IF (NOT(Brusa2_Tx.hton_NoPP_StopTx_Timer.Q) = TRUE) THEN
	ActAC_Rx_Timer(IN := NOT(ActAC_Rx.q_NewData), PT := T#5S);
	ActErr_Rx_Timer(IN := NOT(NLG2_ActErr_Rx.q_NewData), PT := T#5S);
	ActInt_Rx_Timer(IN := NOT(NLG2_ActInt_Rx.q_NewData), PT := T#5S);
	ActLim_Rx_Timer(IN := NOT(NLG2_ActLim_Rx.q_NewData), PT := T#5S);
	ActPlug_Rx_Timer(IN := NOT(NLG2_ActPlug_Rx.q_NewData), PT := T#5S);
	IF (ActAC_Rx_Timer.Q = TRUE AND ActErr_Rx_Timer.Q = TRUE AND ActInt_Rx_Timer.Q = TRUE AND
		ActLim_Rx_Timer.Q = TRUE AND ActPlug_Rx_Timer.Q = TRUE									) THEN
		CommsLoss	:=	TRUE;
	ELSE
		CommsLoss	:=	FALSE;
	END_IF
END_IF

Brusa2_RxConversion();

END_PROGRAM

// Application/UserCode/Brusa/Brusa2_Comms/Brusa2_RxConversion_1
PROGRAM Brusa2_RxConversion_1
VAR
ACVoltL1Act		:	UINT;
	ACVoltL2Act		:	UINT;
	ACVoltL3Act		:	UINT;
	ACCurrL1Act		:	SINT;
	ACCurrL2Act		:	SINT;
	ACCurrL3Act		:	SINT;
	ACPowTotAct		:	UINT;
	MaxTempAct		:	INT;
	TempCon			:	INT;
	DCHVAhAct			:	REAL;
	DCHVVoltAct			:	REAL;
	DCHVCurrAct			:	REAL;
	ACCurrMaxAct		:	REAL;
	ACCurrHWAvl			:	REAL;
	ACCurrMaxCP			:	REAL;
	TempCoolPlate		:	INT;		
END_VAR

ACVoltL1Act	:=	USINT_TO_UINT(Brusa2_Rx.ACVoltL1Act_Rx) * 2;
ACVoltL2Act	:=	USINT_TO_UINT(Brusa2_Rx.ACVoltL2Act_Rx) * 2;
ACVoltL3Act	:=	USINT_TO_UINT(Brusa2_Rx.ACVoltL3Act_Rx) * 2;
ACCurrL1Act	:=	USINT_TO_SINT(Brusa2_Rx.ACCurrL1Act_Rx) - 127;
ACCurrL2Act	:=	USINT_TO_SINT(Brusa2_Rx.ACCurrL2Act_Rx) - 127;
ACCurrL3Act	:=	USINT_TO_SINT(Brusa2_Rx.ACCurrL3Act_Rx) - 127;
ACPowTotAct	:=	USINT_TO_UINT(Brusa2_Rx.ACPowTotAct_Rx) * 100;
MaxTempAct	:=	USINT_TO_INT(Brusa2_Rx.MaxTempAct_Rx) - 50;
TempCon		:=	USINT_TO_INT(Brusa2_Rx.TempCon_Rx) - 50;
DCHVAhAct		:=	UINT_TO_REAL(Brusa2_Rx.DCHVAhAct_Rx) * 0.01;
DCHVVoltAct		:=	UINT_TO_REAL(Brusa2_Rx.DCHVVoltAct_Rx) * 0.1;
DCHVCurrAct		:=	UINT_TO_REAL(Brusa2_Rx.DCHVCurrAct_Rx) * 0.1 - 100;
ACCurrMaxAct	:=	UINT_TO_REAL(Brusa2_Rx.ACCurrMaxAct_Rx) * 0.1 -100;
ACCurrHWAvl		:=	USINT_TO_REAL(Brusa2_Rx.ACCurrHWAvl_Rx) * 0.5;
ACCurrMaxCP		:=	UINT_TO_REAL(Brusa2_Rx.ACCurrMaxCP_Rx) * 0.1;
TempCoolPlate	:=	USINT_TO_INT(Brusa2_Rx.TempCoolPlate_Rx) - 50;

END_PROGRAM

// Application/UserCode/Brusa/Brusa2_Comms/Brusa2_Tx_1
PROGRAM Brusa2_Tx_1

VAR
	DenLim_Tx				:	EPEC_CANVXD.Msg;
	hu8_DenLim_Tx0			:	BYTE;
	hu8_DenLim_Tx2			:	BYTE;
	hu8_DenLim_Tx4			:	BYTE;
	hu8_DenLim_Tx6			:	BYTE;
	hton_Transmit_Timer		:	TON;
	hton_NoPP_StopTx_Timer	:	TON;
	StopBroadcast			:	BOOL;
	C_VentilRq				: 	BOOL;
END_VAR


Brusa2_TxConversion();

StopBroadcast	:=	(NOT(Brusa1_Rx.S_ProximityDet)(* AND DI_q_VehicleKL15_DI = FALSE*));
hton_NoPP_StopTx_Timer(IN := StopBroadcast, PT := T#1S);

// Brusa2_Control.C_Clr_Err	:= FALSE;
hu8_DenLim_Tx0	:=	UINT_TO_USINT(SHR(Brusa2_TxConversion.DCHVVoltLimMax_Tx, 8)) + SHL(BOOL_TO_USINT(C_VentilRq), 5) +
					SHL(BOOL_TO_USINT(Brusa.S_Unlock), 6) + SHL(BOOL_TO_USINT(Brusa.S_ErrClr), 7);
hu8_DenLim_Tx2	:=	(UINT_TO_USINT(SHR(Brusa2_TxConversion.DCHVCurrLimMax_Tx, 8)) AND 2#00000111) + SHL(Brusa.S_StateDem, 5);
hu8_DenLim_Tx4	:=	(UINT_TO_USINT(SHR(Brusa2_TxConversion.ACCurrLimMax_Tx, 8)) AND 2#00000111) + SHL(Brusa.LEDDem, 4);
//hu8_DenLim_Tx6	:=	(UINT_TO_USINT(SHR(Brusa2_TxConversion.ACPhaseShift_Tx, 8)) AND 2#00001111) + SHL(BOOL_TO_USINT(Brusa2_Rx.C_EnPhaseShift), 4);

DenLim_Tx.ID		:=	16#711;
DenLim_Tx.Data[0]	:=	hu8_DenLim_Tx0;
DenLim_Tx.Data[1]	:=	UINT_TO_USINT(Brusa2_TxConversion.DCHVVoltLimMax_Tx);
DenLim_Tx.Data[2]	:=	hu8_DenLim_Tx2;
DenLim_Tx.Data[3]	:=	UINT_TO_USINT(Brusa2_TxConversion.DCHVCurrLimMax_Tx);
DenLim_Tx.Data[4]	:=	hu8_DenLim_Tx4;
DenLim_Tx.Data[5]	:=	UINT_TO_USINT(Brusa2_TxConversion.ACCurrLimMax_Tx);
DenLim_Tx.Data[6]	:=	hu8_DenLim_Tx6;
DenLim_Tx.Data[7]	:=	UINT_TO_USINT(Brusa2_TxConversion.ACPhaseShift_Tx);
DenLim_Tx.Len		:=	8;



hton_Transmit_Timer(IN := NOT(hton_Transmit_Timer.Q), PT := T#90MS);
IF (hton_Transmit_Timer.Q = TRUE AND NOT(hton_NoPP_StopTx_Timer.Q) = TRUE) THEN
	G_CAN3_Channel.SendMessage(i_pMSG:=ADR(DenLim_Tx));
END_IF

END_PROGRAM

// Application/UserCode/Brusa/Brusa2_Comms/Brusa2_TxConversion_1
PROGRAM Brusa2_TxConversion_1
VAR
		DCHVVoltLimMax_Tx	:	UINT;
		DCHVCurrLimMax_Tx	:	UINT;
		ACCurrLimMax_Tx		:	UINT;
		ACPhaseShift_Tx		:	UINT;
END_VAR

//r2
DCHVVoltLimMax_Tx	:=	REAL_TO_UINT(Brusa.S_DCHVVoltLimMax / 0.1);
DCHVCurrLimMax_Tx	:=	REAL_TO_UINT((Brusa.S_DCHVCurrLimMax - 102.4) / 0.1);
ACCurrLimMax_Tx		:=	REAL_TO_UINT((Brusa.S_ACCurrLimMax - 102.4) / 0.1);
//ACPhaseShift_Tx		:=	REAL_TO_UINT(Brusa2_Control.ACPhaseShift / 0.1);

END_PROGRAM

// Application/UserCode/CAN Function Blocks/CAN1/Callback_Receive_CAN1_1
FUNCTION_BLOCK Callback_Receive_CAN1_1 IMPLEMENTS
EPEC_CANVXD.IReceiveCallback
VAR_INPUT	
END_VAR
VAR_OUTPUT
END_VAR
VAR
END_VAR

METHOD Receive
VAR_INPUT
	(* Pointer to the CAN message *)
	i_pMsg	: POINTER TO EPEC_CANVXD.Msg;
	(* User specific argument. This is set in AddCOBID i_Argument. *)
	i_Argument	: DWORD;
END_VAR
VAR
	t_pRxMessage : POINTER TO t_CANReceive;
END_VAR


t_pRxMessage				:=	i_Argument;
t_pRxMessage^.q_NewDataRxed	:=	TRUE;
t_pRxMessage^.Data			:=	i_pMsg^.Data;
t_pRxMessage^.ID			:=	i_pMsg^.ID;
t_pRxMessage^.Len			:=	i_pMsg^.Len;
END_METHOD

END_FUNCTION_BLOCK

// Application/UserCode/CAN Function Blocks/CAN1/Receive_CAN1_EXD_1
FUNCTION_BLOCK Receive_CAN1_EXD_1
VAR_INPUT
	u32_COBID	:	DWORD;
END_VAR
VAR_OUTPUT
	q_NewData	:	BOOL;
	au8_Data	:	ARRAY [0..7] OF BYTE;
	u8_Length	:	BYTE;
END_VAR
VAR
	hq_Initialise	:	BOOL	:=	FALSE;
	ht_RxMessage	:	t_CANReceive;
	ht_MsgRx		:	Callback_Receive_CAN1;
END_VAR



IF (hq_Initialise = FALSE) THEN
	(*
	(*11 bit*)
	G_CAN1_Channel.AddCOBID(i_CobId := u32_COBID,
							i_itfCallback := ht_RxMessage,
							i_Argument := ADR(ht_RxMessage));
	*)
	(*29 bit*)
	G_CAN1_Channel.AddCOBID(i_CobId := u32_COBID OR EPEC_CANVXD.MASK_29BIT,
							i_itfCallback := ht_MsgRx,
							i_Argument := ADR(ht_RxMessage));
	G_CAN1_Channel.SetMask(i_CobID := u32_COBID OR EPEC_CANVXD.MASK_29BIT, i_Mask := (*16#0CFF0211 OR 16#0C010305 OR*) EPEC_CANVXD.MASK_29BIT);

	hq_Initialise	:=	TRUE;
END_IF


IF (ht_RxMessage.q_NewDataRxed = TRUE) THEN
	au8_Data	:=	ht_RxMessage.Data;
	u8_Length	:=	ht_RxMessage.Len;
	q_NewData	:=	TRUE;
	ht_RxMessage.q_NewDataRxed	:=	FALSE;
ELSE
	q_NewData	:=	FALSE;
END_IF

END_FUNCTION_BLOCK

// Application/UserCode/CAN Function Blocks/CAN1/Receive_CAN1_EXD_28bit_1
FUNCTION_BLOCK Receive_CAN1_EXD_28bit_1
VAR_INPUT
	u32_COBID	:	DWORD;
END_VAR
VAR_OUTPUT
	q_NewData	:	BOOL;
	au8_Data	:	ARRAY [0..7] OF BYTE;
	u8_Length	:	BYTE;
END_VAR
VAR
	hq_Initialise	:	BOOL	:=	FALSE;
	ht_RxMessage	:	t_CANReceive;
	ht_MsgRx		:	Callback_Receive_CAN1;
END_VAR



IF (hq_Initialise = FALSE) THEN
	(*
	(*11 bit*)
	G_CAN1_Channel.AddCOBID(i_CobId := u32_COBID,
							i_itfCallback := ht_RxMessage,
							i_Argument := ADR(ht_RxMessage));
	*)
	(*29 bit*)
	G_CAN1_Channel.AddCOBID(i_CobId := u32_COBID OR EPEC_CANVXD.MASK_29BIT,
							i_itfCallback := ht_MsgRx,
							i_Argument := ADR(ht_RxMessage));
	G_CAN1_Channel.SetMask(i_CobID := u32_COBID OR EPEC_CANVXD.MASK_29BIT, i_Mask := 16#0CFF0211 OR 16#0C010305 (*OR EPEC_CANVXD.MASK_29BIT*));

	hq_Initialise	:=	TRUE;
END_IF


IF (ht_RxMessage.q_NewDataRxed = TRUE) THEN
	au8_Data	:=	ht_RxMessage.Data;
	u8_Length	:=	ht_RxMessage.Len;
	q_NewData	:=	TRUE;
	ht_RxMessage.q_NewDataRxed	:=	FALSE;
ELSE
	q_NewData	:=	FALSE;
END_IF

END_FUNCTION_BLOCK

// Application/UserCode/CAN Function Blocks/CAN1/Receive_CAN1_STD_1
FUNCTION_BLOCK Receive_CAN1_STD_1
VAR_INPUT
	u32_COBID	:	DWORD;
END_VAR
VAR_OUTPUT
	q_NewData	:	BOOL;
	au8_Data	:	ARRAY [0..7] OF BYTE;
	u8_Length	:	BYTE;
END_VAR
VAR
	hq_Initialise	:	BOOL	:=	FALSE;
	ht_RxMessage	:	t_CANReceive;
	ht_MsgRx		:	Callback_Receive_CAN1;
END_VAR



IF (hq_Initialise = FALSE) THEN
	
	(*11 bit*)
	G_CAN1_Channel.AddCOBID(i_CobId := u32_COBID,
							i_itfCallback := ht_MsgRx,
							i_Argument := ADR(ht_RxMessage));
	(*
	(*29 bit*)
	G_CAN1_Channel.AddCOBID(i_CobId := u32_COBID OR EPEC_CANVXD.MASK_29BIT,
							i_itfCallback := ht_MsgRx,
							i_Argument := ADR(ht_RxMessage));
*)	(*G_CAN1_Channel.SetMask(i_CobID := u32_COBID OR EPEC_CANVXD.MASK_29BIT, i_Mask := 16#0C009000 OR EPEC_CANVXD.MASK_29BIT);
*)
	hq_Initialise	:=	TRUE;
END_IF


IF (ht_RxMessage.q_NewDataRxed = TRUE) THEN
	au8_Data	:=	ht_RxMessage.Data;
	u8_Length	:=	ht_RxMessage.Len;
	q_NewData	:=	TRUE;
	ht_RxMessage.q_NewDataRxed	:=	FALSE;
ELSE
	q_NewData	:=	FALSE;
END_IF

END_FUNCTION_BLOCK

// Application/UserCode/CAN Function Blocks/CAN2/Callback_Receive_CAN2_1
FUNCTION_BLOCK Callback_Receive_CAN2_1 IMPLEMENTS
EPEC_CANVXD.IReceiveCallback
VAR_INPUT	
END_VAR
VAR_OUTPUT
END_VAR
VAR
END_VAR

METHOD Receive
VAR_INPUT
	(* Pointer to the CAN message *)
	i_pMsg	: POINTER TO EPEC_CANVXD.Msg;
	(* User specific argument. This is set in AddCOBID i_Argument. *)
	i_Argument	: DWORD;
END_VAR
VAR
	t_pRxMessage : POINTER TO t_CANReceive;
END_VAR


t_pRxMessage				:=	i_Argument;
t_pRxMessage^.q_NewDataRxed	:=	TRUE;
t_pRxMessage^.Data			:=	i_pMsg^.Data;
t_pRxMessage^.ID			:=	i_pMsg^.ID;
t_pRxMessage^.Len			:=	i_pMsg^.Len;
END_METHOD

END_FUNCTION_BLOCK

// Application/UserCode/CAN Function Blocks/CAN2/Receive_CAN2_EXD_1
FUNCTION_BLOCK Receive_CAN2_EXD_1
VAR_INPUT
	u32_COBID	:	DWORD;
END_VAR
VAR_OUTPUT
	q_NewData	:	BOOL;
	au8_Data	:	ARRAY [0..7] OF BYTE;
	u8_Length	:	BYTE;
END_VAR
VAR
	hq_Initialise	:	BOOL	:=	FALSE;
	ht_RxMessage	:	t_CANReceive;
	ht_MsgRx		:	Callback_Receive_CAN1;
END_VAR



IF (hq_Initialise = FALSE) THEN
	(*
	IF (u32_COBID > 16#7FF) THEN
		(*29 bit*)
		;
	ELSE
		(*11 bit*)
		;
	END_IF
	*)
	(*
	(*11 bit*)
	G_CAN2_Channel.AddCOBID(i_CobId := u32_COBID,
							i_itfCallback := ht_RxMessage,
							i_Argument := ADR(ht_RxMessage));
	*)
	(*29 bit*)
	G_CAN2_Channel.AddCOBID(i_CobId := u32_COBID OR EPEC_CANVXD.MASK_29BIT,
							i_itfCallback := ht_MsgRx,
							i_Argument := ADR(ht_RxMessage));
	(*G_CAN2_Channel.SetMask(i_CobID := u32_COBID OR EPEC_CANVXD.MASK_29BIT, i_Mask := 16#0C009000 OR EPEC_CANVXD.MASK_29BIT);
*)
	hq_Initialise	:=	TRUE;
END_IF


IF (ht_RxMessage.q_NewDataRxed = TRUE) THEN
	au8_Data	:=	ht_RxMessage.Data;
	u8_Length	:=	ht_RxMessage.Len;
	q_NewData	:=	TRUE;
	ht_RxMessage.q_NewDataRxed	:=	FALSE;
ELSE
	q_NewData	:=	FALSE;
END_IF

END_FUNCTION_BLOCK

// Application/UserCode/CAN Function Blocks/CAN2/Receive_CAN2_STD_1
FUNCTION_BLOCK Receive_CAN2_STD_1
VAR_INPUT
	u32_COBID	:	DWORD;
END_VAR
VAR_OUTPUT
	q_NewData	:	BOOL;
	au8_Data	:	ARRAY [0..7] OF BYTE;
	u8_Length	:	BYTE;
END_VAR
VAR
	hq_Initialise	:	BOOL	:=	FALSE;
	ht_RxMessage	:	t_CANReceive;
	ht_MsgRx		:	Callback_Receive_CAN1;
END_VAR



IF (hq_Initialise = FALSE) THEN
	(*
	IF (u32_COBID > 16#7FF) THEN
		(*29 bit*)
		;
	ELSE
		(*11 bit*)
		;
	END_IF
	*)
	
	(*11 bit*)
	G_CAN2_Channel.AddCOBID(i_CobId := u32_COBID,
							i_itfCallback := ht_MsgRx,
							i_Argument := ADR(ht_RxMessage));
	(*
	(*29 bit*)
	G_CAN2_Channel.AddCOBID(i_CobId := u32_COBID OR EPEC_CANVXD.MASK_29BIT,
							i_itfCallback := ht_MsgRx,
							i_Argument := ADR(ht_RxMessage));
*)	(*G_CAN2_Channel.SetMask(i_CobID := u32_COBID OR EPEC_CANVXD.MASK_29BIT, i_Mask := 16#0C009000 OR EPEC_CANVXD.MASK_29BIT);
*)
	hq_Initialise	:=	TRUE;
END_IF


IF (ht_RxMessage.q_NewDataRxed = TRUE) THEN
	au8_Data	:=	ht_RxMessage.Data;
	u8_Length	:=	ht_RxMessage.Len;
	q_NewData	:=	TRUE;
	ht_RxMessage.q_NewDataRxed	:=	FALSE;
ELSE
	q_NewData	:=	FALSE;
END_IF

END_FUNCTION_BLOCK

// Application/UserCode/CAN Function Blocks/CAN3/Callback_Receive_CAN3_1
FUNCTION_BLOCK Callback_Receive_CAN3_1 IMPLEMENTS
EPEC_CANVXD.IReceiveCallback
VAR_INPUT	
END_VAR
VAR_OUTPUT
END_VAR
VAR
END_VAR

METHOD Receive
VAR_INPUT
	(* Pointer to the CAN message *)
	i_pMsg	: POINTER TO EPEC_CANVXD.Msg;
	(* User specific argument. This is set in AddCOBID i_Argument. *)
	i_Argument	: DWORD;
END_VAR
VAR
	t_pRxMessage : POINTER TO t_CANReceive;
END_VAR


t_pRxMessage				:=	i_Argument;
t_pRxMessage^.q_NewDataRxed	:=	TRUE;
t_pRxMessage^.Data			:=	i_pMsg^.Data;
t_pRxMessage^.ID			:=	i_pMsg^.ID;
t_pRxMessage^.Len			:=	i_pMsg^.Len;
END_METHOD

END_FUNCTION_BLOCK

// Application/UserCode/CAN Function Blocks/CAN3/Receive_CAN3_EXD_1
FUNCTION_BLOCK Receive_CAN3_EXD_1
VAR_INPUT
	u32_COBID	:	DWORD;
END_VAR
VAR_OUTPUT
	q_NewData	:	BOOL;
	au8_Data	:	ARRAY [0..7] OF BYTE;
	u8_Length	:	BYTE;
END_VAR
VAR
	hq_Initialise	:	BOOL	:=	FALSE;
	ht_RxMessage	:	t_CANReceive;
	ht_MsgRx		:	Callback_Receive_CAN1;
END_VAR



IF (hq_Initialise = FALSE) THEN
	(*
	IF (u32_COBID > 16#7FF) THEN
		(*29 bit*)
		;
	ELSE
		(*11 bit*)
		;
	END_IF
	*)
	(*
	(*11 bit*)
	G_CAN3_Channel.AddCOBID(i_CobId := u32_COBID,
							i_itfCallback := ht_RxMessage,
							i_Argument := ADR(ht_RxMessage));
	*)
	(*29 bit*)
	G_CAN3_Channel.AddCOBID(i_CobId := u32_COBID OR EPEC_CANVXD.MASK_29BIT,
							i_itfCallback := ht_MsgRx,
							i_Argument := ADR(ht_RxMessage));
	G_CAN3_Channel.SetMask(i_CobID := u32_COBID OR EPEC_CANVXD.MASK_29BIT, (*i_Mask := 16#0C009000 OR*) EPEC_CANVXD.MASK_29BIT);

	hq_Initialise	:=	TRUE;
END_IF


IF (ht_RxMessage.q_NewDataRxed = TRUE) THEN
	au8_Data	:=	ht_RxMessage.Data;
	u8_Length	:=	ht_RxMessage.Len;
	q_NewData	:=	TRUE;
	ht_RxMessage.q_NewDataRxed	:=	FALSE;
ELSE
	q_NewData	:=	FALSE;
END_IF

END_FUNCTION_BLOCK

// Application/UserCode/CAN Function Blocks/CAN3/Receive_CAN3_EXD_28bit_1
FUNCTION_BLOCK Receive_CAN3_EXD_28bit_1
VAR_INPUT
	u32_COBID	:	DWORD;
END_VAR
VAR_OUTPUT
	q_NewData	:	BOOL;
	au8_Data	:	ARRAY [0..7] OF BYTE;
	u8_Length	:	BYTE;
END_VAR
VAR
	hq_Initialise	:	BOOL	:=	FALSE;
	ht_RxMessage	:	t_CANReceive;
	ht_MsgRx		:	Callback_Receive_CAN1;
END_VAR



IF (hq_Initialise = FALSE) THEN
	(*
	IF (u32_COBID > 16#7FF) THEN
		(*29 bit*)
		;
	ELSE
		(*11 bit*)
		;
	END_IF
	*)
	(*
	(*11 bit*)
	G_CAN3_Channel.AddCOBID(i_CobId := u32_COBID,
							i_itfCallback := ht_RxMessage,
							i_Argument := ADR(ht_RxMessage));
	*)
	(*29 bit*)
	G_CAN3_Channel.AddCOBID(i_CobId := u32_COBID OR EPEC_CANVXD.MASK_29BIT,
							i_itfCallback := ht_MsgRx,
							i_Argument := ADR(ht_RxMessage));
	G_CAN3_Channel.SetMask(i_CobID := u32_COBID OR EPEC_CANVXD.MASK_29BIT, i_Mask := 16#0C010305);

	hq_Initialise	:=	TRUE;
END_IF


IF (ht_RxMessage.q_NewDataRxed = TRUE) THEN
	au8_Data	:=	ht_RxMessage.Data;
	u8_Length	:=	ht_RxMessage.Len;
	q_NewData	:=	TRUE;
	ht_RxMessage.q_NewDataRxed	:=	FALSE;
ELSE
	q_NewData	:=	FALSE;
END_IF

END_FUNCTION_BLOCK

// Application/UserCode/CAN Function Blocks/CAN3/Receive_CAN3_STD_1
FUNCTION_BLOCK Receive_CAN3_STD_1
VAR_INPUT
	u32_COBID	:	DWORD;
END_VAR
VAR_OUTPUT
	q_NewData	:	BOOL;
	au8_Data	:	ARRAY [0..7] OF BYTE;
	u8_Length	:	BYTE;
END_VAR
VAR
	hq_Initialise	:	BOOL	:=	FALSE;
	ht_RxMessage	:	t_CANReceive;
	ht_MsgRx		:	Callback_Receive_CAN1;
END_VAR



IF (hq_Initialise = FALSE) THEN
	(*
	IF (u32_COBID > 16#7FF) THEN
		(*29 bit*)
		;
	ELSE
		(*11 bit*)
		;
	END_IF
	*)
	
	(*11 bit*)
	G_CAN3_Channel.AddCOBID(i_CobId := u32_COBID,
							i_itfCallback := ht_MsgRx,
							i_Argument := ADR(ht_RxMessage));
	(*
	(*29 bit*)
	G_CAN3_Channel.AddCOBID(i_CobId := u32_COBID OR EPEC_CANVXD.MASK_29BIT,
							i_itfCallback := ht_MsgRx,
							i_Argument := ADR(ht_RxMessage));
*)	(*G_CAN3_Channel.SetMask(i_CobID := u32_COBID OR EPEC_CANVXD.MASK_29BIT, i_Mask := 16#0C009000 OR EPEC_CANVXD.MASK_29BIT);
*)
	hq_Initialise	:=	TRUE;
END_IF


IF (ht_RxMessage.q_NewDataRxed = TRUE) THEN
	au8_Data	:=	ht_RxMessage.Data;
	u8_Length	:=	ht_RxMessage.Len;
	q_NewData	:=	TRUE;
	ht_RxMessage.q_NewDataRxed	:=	FALSE;
ELSE
	q_NewData	:=	FALSE;
END_IF

END_FUNCTION_BLOCK

// Application/UserCode/CAN Function Blocks/CAN4/Callback_Receive_CAN4_1
FUNCTION_BLOCK Callback_Receive_CAN4_1 IMPLEMENTS
EPEC_CANVXD.IReceiveCallback
VAR_INPUT	
END_VAR
VAR_OUTPUT
END_VAR
VAR
END_VAR

METHOD Receive
VAR_INPUT
	(* Pointer to the CAN message *)
	i_pMsg	: POINTER TO EPEC_CANVXD.Msg;
	(* User specific argument. This is set in AddCOBID i_Argument. *)
	i_Argument	: DWORD;
END_VAR
VAR
	t_pRxMessage : POINTER TO t_CANReceive;
END_VAR


t_pRxMessage				:=	i_Argument;
t_pRxMessage^.q_NewDataRxed	:=	TRUE;
t_pRxMessage^.Data			:=	i_pMsg^.Data;
t_pRxMessage^.ID			:=	i_pMsg^.ID;
t_pRxMessage^.Len			:=	i_pMsg^.Len;
END_METHOD

END_FUNCTION_BLOCK

// Application/UserCode/CAN Function Blocks/CAN4/Receive_CAN4_EXD_1
FUNCTION_BLOCK Receive_CAN4_EXD_1
VAR_INPUT
	u32_COBID	:	DWORD;
END_VAR
VAR_OUTPUT
	q_NewData	:	BOOL;
	au8_Data	:	ARRAY [0..7] OF BYTE;
	u8_Length	:	BYTE;
END_VAR
VAR
	hq_Initialise	:	BOOL	:=	FALSE;
	ht_RxMessage	:	t_CANReceive;
	ht_MsgRx		:	Callback_Receive_CAN1;
END_VAR



IF (hq_Initialise = FALSE) THEN
	(*
	IF (u32_COBID > 16#7FF) THEN
		(*29 bit*)
		;
	ELSE
		(*11 bit*)
		;
	END_IF
	*)
	(*
	(*11 bit*)
	G_CAN4_Channel.AddCOBID(i_CobId := u32_COBID,
							i_itfCallback := ht_RxMessage,
							i_Argument := ADR(ht_RxMessage));
	*)
	(*29 bit*)
	G_CAN4_Channel.AddCOBID(i_CobId := u32_COBID OR EPEC_CANVXD.MASK_29BIT,
							i_itfCallback := ht_MsgRx,
							i_Argument := ADR(ht_RxMessage));
	G_CAN4_Channel.SetMask(i_CobID := u32_COBID OR EPEC_CANVXD.MASK_29BIT, i_Mask := 16#18FEF1F2 OR EPEC_CANVXD.MASK_29BIT);

	hq_Initialise	:=	TRUE;
END_IF


IF (ht_RxMessage.q_NewDataRxed = TRUE) THEN
	au8_Data	:=	ht_RxMessage.Data;
	u8_Length	:=	ht_RxMessage.Len;
	q_NewData	:=	TRUE;
	ht_RxMessage.q_NewDataRxed	:=	FALSE;
ELSE
	q_NewData	:=	FALSE;
END_IF

END_FUNCTION_BLOCK

// Application/UserCode/CAN Function Blocks/CAN4/Receive_CAN4_STD_1
FUNCTION_BLOCK Receive_CAN4_STD_1
VAR_INPUT
	u32_COBID	:	DWORD;
END_VAR
VAR_OUTPUT
	q_NewData	:	BOOL;
	au8_Data	:	ARRAY [0..7] OF BYTE;
	u8_Length	:	BYTE;
END_VAR
VAR
	hq_Initialise	:	BOOL	:=	FALSE;
	ht_RxMessage	:	t_CANReceive;
	ht_MsgRx		:	Callback_Receive_CAN1;
END_VAR



IF (hq_Initialise = FALSE) THEN
	(*
	IF (u32_COBID > 16#7FF) THEN
		(*29 bit*)
		;
	ELSE
		(*11 bit*)
		;
	END_IF
	*)
	
	(*11 bit*)
	G_CAN4_Channel.AddCOBID(i_CobId := u32_COBID,
							i_itfCallback := ht_MsgRx,
							i_Argument := ADR(ht_RxMessage));
	(*
	(*29 bit*)
	G_CAN4_Channel.AddCOBID(i_CobId := u32_COBID OR EPEC_CANVXD.MASK_29BIT,
							i_itfCallback := ht_MsgRx,
							i_Argument := ADR(ht_RxMessage));
*)	(*G_CAN4_Channel.SetMask(i_CobID := u32_COBID OR EPEC_CANVXD.MASK_29BIT, i_Mask := 16#0C009000 OR EPEC_CANVXD.MASK_29BIT);
*)
	hq_Initialise	:=	TRUE;
END_IF


IF (ht_RxMessage.q_NewDataRxed = TRUE) THEN
	au8_Data	:=	ht_RxMessage.Data;
	u8_Length	:=	ht_RxMessage.Len;
	q_NewData	:=	TRUE;
	ht_RxMessage.q_NewDataRxed	:=	FALSE;
ELSE
	q_NewData	:=	FALSE;
END_IF

END_FUNCTION_BLOCK

// Application/UserCode/Main Program/RealTimeClock
PROGRAM RealTimeClock

VAR
	RTC_0: rtc;
	Timesky: DATE_AND_TIME := DT#2021-10-29-17:31:0;
	today: DATE_AND_TIME;
	a1870: DATE_AND_TIME := DT#1970-1-1-0:0:0;
END_VAR

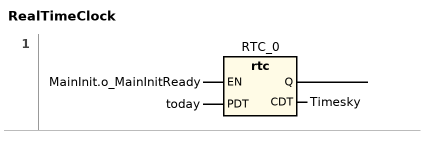
// NETWORK 1
RTC_0(EN := MainInit.o_MainInitReady, PDT := today, CDT => Timesky); // rtc

END_PROGRAM

// Application/UserCode/HMI/Data to or For HMI/BMS_to_HMI_1
PROGRAM BMS_to_HMI_1
VAR
	ht_CAN4_DD0_Tx	:	EPEC_CANVXD.Msg;
	ht_CAN4_DD1_Tx	:	EPEC_CANVXD.Msg;
	ht_CAN4_DD2_Tx	:	EPEC_CANVXD.Msg;
	ht_CAN4_DD3_Tx	:	EPEC_CANVXD.Msg;
	ht_CAN4_DD4_Tx	:	EPEC_CANVXD.Msg;
	ht_CAN4_DD5_Tx	:	EPEC_CANVXD.Msg;
	ht_CAN4_DD6_Tx	:	EPEC_CANVXD.Msg;
	ht_CAN4_DD7_Tx	:	EPEC_CANVXD.Msg;
	ht_CAN4_DD8_Tx	:	EPEC_CANVXD.Msg;
	ht_CAN4_DD9_Tx	:	EPEC_CANVXD.Msg;
	ht_CAN4_DDA_Tx	:	EPEC_CANVXD.Msg;
	ht_CAN4_DDB_Tx	:	EPEC_CANVXD.Msg;
	ht_CAN4_DDC_Tx	:	EPEC_CANVXD.Msg;
	ht_CAN4_DDD_Tx	:	EPEC_CANVXD.Msg;
	ht_CAN4_ADD0_Tx	:	EPEC_CANVXD.Msg;
	ht_CAN4_ADD1_Tx	:	EPEC_CANVXD.Msg;
	ht_CAN4_ADD2_Tx	:	EPEC_CANVXD.Msg;
	ht_CAN4_ADD3_Tx	:	EPEC_CANVXD.Msg;
	ht_CAN4_ADD4_Tx	:	EPEC_CANVXD.Msg;
	ht_CAN4_ADD5_Tx	:	EPEC_CANVXD.Msg;
	ht_CAN4_ADD6_Tx	:	EPEC_CANVXD.Msg;
	ht_CAN4_ADD7_Tx	:	EPEC_CANVXD.Msg;
	ht_CAN4_ADD8_Tx	:	EPEC_CANVXD.Msg;
	ht_CAN4_ADD9_Tx	:	EPEC_CANVXD.Msg;
	ht_CAN4_ADDA_Tx	:	EPEC_CANVXD.Msg;
	ht_CAN4_ADDB_Tx	:	EPEC_CANVXD.Msg;
	ht_CAN4_ADDC_Tx	:	EPEC_CANVXD.Msg;
	ht_CAN4_ADDD_Tx	:	EPEC_CANVXD.Msg;
	hton_MessageSend_Timer	:	TON;
	
	Tx_Timer	:	TON;
	
END_VAR

//Send raw BMS Data to HMI CAN#4
(*BMS1*)
ht_CAN4_DD0_Tx.ID		:=	16#181000DD OR EPEC_CANVXD.MASK_29BIT;
ht_CAN4_DD0_Tx.Data[0]	:=	OrionBMS1_Rx.OrionBMS1_6B0_Rx.au8_Data[0];
ht_CAN4_DD0_Tx.Data[1]	:=	OrionBMS1_Rx.OrionBMS1_6B0_Rx.au8_Data[1];
ht_CAN4_DD0_Tx.Data[2]	:=	OrionBMS1_Rx.OrionBMS1_6B0_Rx.au8_Data[2];
ht_CAN4_DD0_Tx.Data[3]	:=	OrionBMS1_Rx.OrionBMS1_6B0_Rx.au8_Data[3];
ht_CAN4_DD0_Tx.Data[4]	:=	OrionBMS1_Rx.OrionBMS1_6B0_Rx.au8_Data[4];
ht_CAN4_DD0_Tx.Data[5]	:=	OrionBMS1_Rx.OrionBMS1_6B0_Rx.au8_Data[5];		
ht_CAN4_DD0_Tx.Data[6]	:=	OrionBMS1_Rx.OrionBMS1_6B0_Rx.au8_Data[6];	
ht_CAN4_DD0_Tx.Data[7]	:=	OrionBMS1_Rx.OrionBMS1_6B0_Rx.au8_Data[7];		
ht_CAN4_DD0_Tx.Len		:=	8;

ht_CAN4_DD1_Tx.ID		:=	16#181001DD OR EPEC_CANVXD.MASK_29BIT;
ht_CAN4_DD1_Tx.Data[0]	:=	OrionBMS1_Rx.OrionBMS1_6B1_Rx.au8_Data[0];
ht_CAN4_DD1_Tx.Data[1]	:=	OrionBMS1_Rx.OrionBMS1_6B1_Rx.au8_Data[1];
ht_CAN4_DD1_Tx.Data[2]	:=	OrionBMS1_Rx.OrionBMS1_6B1_Rx.au8_Data[2];
ht_CAN4_DD1_Tx.Data[3]	:=	OrionBMS1_Rx.OrionBMS1_6B1_Rx.au8_Data[3];
ht_CAN4_DD1_Tx.Data[4]	:=	OrionBMS1_Rx.OrionBMS1_6B1_Rx.au8_Data[4];
ht_CAN4_DD1_Tx.Data[5]	:=	OrionBMS1_Rx.OrionBMS1_6B1_Rx.au8_Data[5];		
ht_CAN4_DD1_Tx.Data[6]	:=	OrionBMS1_Rx.OrionBMS1_6B1_Rx.au8_Data[6];	
ht_CAN4_DD1_Tx.Data[7]	:=	OrionBMS1_Rx.OrionBMS1_6B1_Rx.au8_Data[7];		
ht_CAN4_DD1_Tx.Len		:=	8;

ht_CAN4_DD2_Tx.ID		:=	16#181002DD OR EPEC_CANVXD.MASK_29BIT;
ht_CAN4_DD2_Tx.Data[0]	:=	OrionBMS1_Rx.OrionBMS1_6B2_Rx.au8_Data[0];
ht_CAN4_DD2_Tx.Data[1]	:=	OrionBMS1_Rx.OrionBMS1_6B2_Rx.au8_Data[1];
ht_CAN4_DD2_Tx.Data[2]	:=	OrionBMS1_Rx.OrionBMS1_6B2_Rx.au8_Data[2];
ht_CAN4_DD2_Tx.Data[3]	:=	OrionBMS1_Rx.OrionBMS1_6B2_Rx.au8_Data[3];
ht_CAN4_DD2_Tx.Data[4]	:=	OrionBMS1_Rx.OrionBMS1_6B2_Rx.au8_Data[4];
ht_CAN4_DD2_Tx.Data[5]	:=	OrionBMS1_Rx.OrionBMS1_6B2_Rx.au8_Data[5];		
ht_CAN4_DD2_Tx.Data[6]	:=	OrionBMS1_Rx.OrionBMS1_6B2_Rx.au8_Data[6];	
ht_CAN4_DD2_Tx.Data[7]	:=	OrionBMS1_Rx.OrionBMS1_6B2_Rx.au8_Data[7];		
ht_CAN4_DD2_Tx.Len		:=	8;

ht_CAN4_DD3_Tx.ID		:=	16#181003DD OR EPEC_CANVXD.MASK_29BIT;
ht_CAN4_DD3_Tx.Data[0]	:=	OrionBMS1_Rx.OrionBMS1_6B3_Rx.au8_Data[0];
ht_CAN4_DD3_Tx.Data[1]	:=	OrionBMS1_Rx.OrionBMS1_6B3_Rx.au8_Data[1];
ht_CAN4_DD3_Tx.Data[2]	:=	OrionBMS1_Rx.OrionBMS1_6B3_Rx.au8_Data[2];
ht_CAN4_DD3_Tx.Data[3]	:=	OrionBMS1_Rx.OrionBMS1_6B3_Rx.au8_Data[3];
ht_CAN4_DD3_Tx.Data[4]	:=	OrionBMS1_Rx.OrionBMS1_6B3_Rx.au8_Data[4];
ht_CAN4_DD3_Tx.Data[5]	:=	OrionBMS1_Rx.OrionBMS1_6B3_Rx.au8_Data[5];		
ht_CAN4_DD3_Tx.Data[6]	:=	OrionBMS1_Rx.OrionBMS1_6B3_Rx.au8_Data[6];	
ht_CAN4_DD3_Tx.Data[7]	:=	OrionBMS1_Rx.OrionBMS1_6B3_Rx.au8_Data[7];		
ht_CAN4_DD3_Tx.Len		:=	8;

ht_CAN4_DD4_Tx.ID		:=	16#181004DD OR EPEC_CANVXD.MASK_29BIT;
ht_CAN4_DD4_Tx.Data[0]	:=	OrionBMS1_Rx.OrionBMS1_6B4_Rx.au8_Data[0];
ht_CAN4_DD4_Tx.Data[1]	:=	OrionBMS1_Rx.OrionBMS1_6B4_Rx.au8_Data[1];
ht_CAN4_DD4_Tx.Data[2]	:=	OrionBMS1_Rx.OrionBMS1_6B4_Rx.au8_Data[2];
ht_CAN4_DD4_Tx.Data[3]	:=	OrionBMS1_Rx.OrionBMS1_6B4_Rx.au8_Data[3];
ht_CAN4_DD4_Tx.Data[4]	:=	OrionBMS1_Rx.OrionBMS1_6B4_Rx.au8_Data[4];
ht_CAN4_DD4_Tx.Data[5]	:=	OrionBMS1_Rx.OrionBMS1_6B4_Rx.au8_Data[5];		
ht_CAN4_DD4_Tx.Data[6]	:=	OrionBMS1_Rx.OrionBMS1_6B4_Rx.au8_Data[6];	
ht_CAN4_DD4_Tx.Data[7]	:=	OrionBMS1_Rx.OrionBMS1_6B4_Rx.au8_Data[7];		
ht_CAN4_DD4_Tx.Len		:=	8;

ht_CAN4_DD5_Tx.ID		:=	16#181005DD OR EPEC_CANVXD.MASK_29BIT;
ht_CAN4_DD5_Tx.Data[0]	:=	OrionBMS1_Rx.OrionBMS1_6B5_Rx.au8_Data[0];
ht_CAN4_DD5_Tx.Data[1]	:=	OrionBMS1_Rx.OrionBMS1_6B5_Rx.au8_Data[1];
ht_CAN4_DD5_Tx.Data[2]	:=	OrionBMS1_Rx.OrionBMS1_6B5_Rx.au8_Data[2];
ht_CAN4_DD5_Tx.Data[3]	:=	OrionBMS1_Rx.OrionBMS1_6B5_Rx.au8_Data[3];
ht_CAN4_DD5_Tx.Data[4]	:=	OrionBMS1_Rx.OrionBMS1_6B5_Rx.au8_Data[4];
ht_CAN4_DD5_Tx.Data[5]	:=	OrionBMS1_Rx.OrionBMS1_6B5_Rx.au8_Data[5];		
ht_CAN4_DD5_Tx.Data[6]	:=	OrionBMS1_Rx.OrionBMS1_6B5_Rx.au8_Data[6];	
ht_CAN4_DD5_Tx.Data[7]	:=	OrionBMS1_Rx.OrionBMS1_6B5_Rx.au8_Data[7];		
ht_CAN4_DD5_Tx.Len		:=	8;

ht_CAN4_DD6_Tx.ID		:=	16#181006DD OR EPEC_CANVXD.MASK_29BIT;
ht_CAN4_DD6_Tx.Data[0]	:=	OrionBMS1_Rx.OrionBMS1_6B6_Rx.au8_Data[0];
ht_CAN4_DD6_Tx.Data[1]	:=	OrionBMS1_Rx.OrionBMS1_6B6_Rx.au8_Data[1];
ht_CAN4_DD6_Tx.Data[2]	:=	OrionBMS1_Rx.OrionBMS1_6B6_Rx.au8_Data[2];
ht_CAN4_DD6_Tx.Data[3]	:=	OrionBMS1_Rx.OrionBMS1_6B6_Rx.au8_Data[3];
ht_CAN4_DD6_Tx.Data[4]	:=	OrionBMS1_Rx.OrionBMS1_6B6_Rx.au8_Data[4];
ht_CAN4_DD6_Tx.Data[5]	:=	OrionBMS1_Rx.OrionBMS1_6B6_Rx.au8_Data[5];		
ht_CAN4_DD6_Tx.Data[6]	:=	OrionBMS1_Rx.OrionBMS1_6B6_Rx.au8_Data[6];	
ht_CAN4_DD6_Tx.Data[7]	:=	OrionBMS1_Rx.OrionBMS1_6B6_Rx.au8_Data[7];		
ht_CAN4_DD6_Tx.Len		:=	8;

ht_CAN4_DD7_Tx.ID		:=	16#181007DD OR EPEC_CANVXD.MASK_29BIT;
ht_CAN4_DD7_Tx.Data[0]	:=	OrionBMS1_Rx.OrionBMS1_6B7_Rx.au8_Data[0];
ht_CAN4_DD7_Tx.Data[1]	:=	OrionBMS1_Rx.OrionBMS1_6B7_Rx.au8_Data[1];
ht_CAN4_DD7_Tx.Data[2]	:=	OrionBMS1_Rx.OrionBMS1_6B7_Rx.au8_Data[2];
ht_CAN4_DD7_Tx.Data[3]	:=	OrionBMS1_Rx.OrionBMS1_6B7_Rx.au8_Data[3];
ht_CAN4_DD7_Tx.Data[4]	:=	OrionBMS1_Rx.OrionBMS1_6B7_Rx.au8_Data[4];
ht_CAN4_DD7_Tx.Data[5]	:=	OrionBMS1_Rx.OrionBMS1_6B7_Rx.au8_Data[5];		
ht_CAN4_DD7_Tx.Data[6]	:=	OrionBMS1_Rx.OrionBMS1_6B7_Rx.au8_Data[6];	
ht_CAN4_DD7_Tx.Data[7]	:=	OrionBMS1_Rx.OrionBMS1_6B7_Rx.au8_Data[7];		
ht_CAN4_DD7_Tx.Len		:=	8;

ht_CAN4_DD8_Tx.ID		:=	16#181008DD OR EPEC_CANVXD.MASK_29BIT;
ht_CAN4_DD8_Tx.Data[0]	:=	OrionBMS1_Rx.OrionBMS1_6B8_Rx.au8_Data[0];
ht_CAN4_DD8_Tx.Data[1]	:=	OrionBMS1_Rx.OrionBMS1_6B8_Rx.au8_Data[1];
ht_CAN4_DD8_Tx.Data[2]	:=	OrionBMS1_Rx.OrionBMS1_6B8_Rx.au8_Data[2];
ht_CAN4_DD8_Tx.Data[3]	:=	OrionBMS1_Rx.OrionBMS1_6B8_Rx.au8_Data[3];
ht_CAN4_DD8_Tx.Data[4]	:=	OrionBMS1_Rx.OrionBMS1_6B8_Rx.au8_Data[4];
ht_CAN4_DD8_Tx.Data[5]	:=	OrionBMS1_Rx.OrionBMS1_6B8_Rx.au8_Data[5];		
ht_CAN4_DD8_Tx.Data[6]	:=	OrionBMS1_Rx.OrionBMS1_6B8_Rx.au8_Data[6];	
ht_CAN4_DD8_Tx.Data[7]	:=	OrionBMS1_Rx.OrionBMS1_6B8_Rx.au8_Data[7];		
ht_CAN4_DD8_Tx.Len		:=	8;

ht_CAN4_DD9_Tx.ID		:=	16#181009DD OR EPEC_CANVXD.MASK_29BIT;
ht_CAN4_DD9_Tx.Data[0]	:=	OrionBMS1_Rx.OrionBMS1_6B9_Rx.au8_Data[0];
ht_CAN4_DD9_Tx.Data[1]	:=	OrionBMS1_Rx.OrionBMS1_6B9_Rx.au8_Data[1];
ht_CAN4_DD9_Tx.Data[2]	:=	OrionBMS1_Rx.OrionBMS1_6B9_Rx.au8_Data[2];
ht_CAN4_DD9_Tx.Data[3]	:=	OrionBMS1_Rx.OrionBMS1_6B9_Rx.au8_Data[3];
ht_CAN4_DD9_Tx.Data[4]	:=	OrionBMS1_Rx.OrionBMS1_6B9_Rx.au8_Data[4];
ht_CAN4_DD9_Tx.Data[5]	:=	OrionBMS1_Rx.OrionBMS1_6B9_Rx.au8_Data[5];		
ht_CAN4_DD9_Tx.Data[6]	:=	OrionBMS1_Rx.OrionBMS1_6B9_Rx.au8_Data[6];	
ht_CAN4_DD9_Tx.Data[7]	:=	OrionBMS1_Rx.OrionBMS1_6B9_Rx.au8_Data[7];		
ht_CAN4_DD9_Tx.Len		:=	8;

ht_CAN4_DDA_Tx.ID		:=	16#18100ADD OR EPEC_CANVXD.MASK_29BIT;
ht_CAN4_DDA_Tx.Data[0]	:=	OrionBMS1_Rx.OrionBMS1_6BA_Rx.au8_Data[0];
ht_CAN4_DDA_Tx.Data[1]	:=	OrionBMS1_Rx.OrionBMS1_6BA_Rx.au8_Data[1];
ht_CAN4_DDA_Tx.Data[2]	:=	OrionBMS1_Rx.OrionBMS1_6BA_Rx.au8_Data[2];
ht_CAN4_DDA_Tx.Data[3]	:=	OrionBMS1_Rx.OrionBMS1_6BA_Rx.au8_Data[3];
ht_CAN4_DDA_Tx.Data[4]	:=	OrionBMS1_Rx.OrionBMS1_6BA_Rx.au8_Data[4];
ht_CAN4_DDA_Tx.Data[5]	:=	OrionBMS1_Rx.OrionBMS1_6BA_Rx.au8_Data[5];		
ht_CAN4_DDA_Tx.Data[6]	:=	OrionBMS1_Rx.OrionBMS1_6BA_Rx.au8_Data[6];	
ht_CAN4_DDA_Tx.Data[7]	:=	OrionBMS1_Rx.OrionBMS1_6BA_Rx.au8_Data[7];		
ht_CAN4_DDA_Tx.Len		:=	8;

ht_CAN4_DDB_Tx.ID		:=	16#18100BDD OR EPEC_CANVXD.MASK_29BIT;
ht_CAN4_DDB_Tx.Data[0]	:=	OrionBMS1_Rx.OrionBMS1_6BB_Rx.au8_Data[0];
ht_CAN4_DDB_Tx.Data[1]	:=	OrionBMS1_Rx.OrionBMS1_6BB_Rx.au8_Data[1];
ht_CAN4_DDB_Tx.Data[2]	:=	OrionBMS1_Rx.OrionBMS1_6BB_Rx.au8_Data[2];
ht_CAN4_DDB_Tx.Data[3]	:=	OrionBMS1_Rx.OrionBMS1_6BB_Rx.au8_Data[3];
ht_CAN4_DDB_Tx.Data[4]	:=	OrionBMS1_Rx.OrionBMS1_6BB_Rx.au8_Data[4];
ht_CAN4_DDB_Tx.Data[5]	:=	OrionBMS1_Rx.OrionBMS1_6BB_Rx.au8_Data[5];		
ht_CAN4_DDB_Tx.Data[6]	:=	OrionBMS1_Rx.OrionBMS1_6BB_Rx.au8_Data[6];	
ht_CAN4_DDB_Tx.Data[7]	:=	OrionBMS1_Rx.OrionBMS1_6BB_Rx.au8_Data[7];		
ht_CAN4_DDB_Tx.Len		:=	8;

ht_CAN4_DDC_Tx.ID		:=	16#18100CDD OR EPEC_CANVXD.MASK_29BIT;
ht_CAN4_DDC_Tx.Data[0]	:=	OrionBMS1_Rx.OrionBMS1_6BC_Rx.au8_Data[0];
ht_CAN4_DDC_Tx.Data[1]	:=	OrionBMS1_Rx.OrionBMS1_6BC_Rx.au8_Data[1];
ht_CAN4_DDC_Tx.Data[2]	:=	OrionBMS1_Rx.OrionBMS1_6BC_Rx.au8_Data[2];
ht_CAN4_DDC_Tx.Data[3]	:=	OrionBMS1_Rx.OrionBMS1_6BC_Rx.au8_Data[3];
ht_CAN4_DDC_Tx.Data[4]	:=	OrionBMS1_Rx.OrionBMS1_6BC_Rx.au8_Data[4];
ht_CAN4_DDC_Tx.Data[5]	:=	OrionBMS1_Rx.OrionBMS1_6BC_Rx.au8_Data[5];		
ht_CAN4_DDC_Tx.Data[6]	:=	OrionBMS1_Rx.OrionBMS1_6BC_Rx.au8_Data[6];	
ht_CAN4_DDC_Tx.Data[7]	:=	OrionBMS1_Rx.OrionBMS1_6BC_Rx.au8_Data[7];		
ht_CAN4_DDC_Tx.Len		:=	8;

ht_CAN4_DDD_Tx.ID		:=	16#18100DDD OR EPEC_CANVXD.MASK_29BIT;
ht_CAN4_DDD_Tx.Data[0]	:=	OrionBMS1_Rx.OrionBMS1_6BD_Rx.au8_Data[0];
ht_CAN4_DDD_Tx.Data[1]	:=	OrionBMS1_Rx.OrionBMS1_6BD_Rx.au8_Data[1];
ht_CAN4_DDD_Tx.Data[2]	:=	OrionBMS1_Rx.OrionBMS1_6BD_Rx.au8_Data[2];
ht_CAN4_DDD_Tx.Data[3]	:=	OrionBMS1_Rx.OrionBMS1_6BD_Rx.au8_Data[3];
ht_CAN4_DDD_Tx.Data[4]	:=	OrionBMS1_Rx.OrionBMS1_6BD_Rx.au8_Data[4];
ht_CAN4_DDD_Tx.Data[5]	:=	OrionBMS1_Rx.OrionBMS1_6BD_Rx.au8_Data[5];		
ht_CAN4_DDD_Tx.Data[6]	:=	OrionBMS1_Rx.OrionBMS1_6BD_Rx.au8_Data[6];	
ht_CAN4_DDD_Tx.Data[7]	:=	OrionBMS1_Rx.OrionBMS1_6BD_Rx.au8_Data[7];		
ht_CAN4_DDD_Tx.Len		:=	8;

//*BMS Slave
ht_CAN4_ADD0_Tx.ID		:=	16#182000DD OR EPEC_CANVXD.MASK_29BIT;
ht_CAN4_ADD0_Tx.Data[0]	:=	OrionBMS2_Rx.OrionBMS2_6B0_Rx.au8_Data[0];
ht_CAN4_ADD0_Tx.Data[1]	:=	OrionBMS2_Rx.OrionBMS2_6B0_Rx.au8_Data[1];
ht_CAN4_ADD0_Tx.Data[2]	:=	OrionBMS2_Rx.OrionBMS2_6B0_Rx.au8_Data[2];
ht_CAN4_ADD0_Tx.Data[3]	:=	OrionBMS2_Rx.OrionBMS2_6B0_Rx.au8_Data[3];
ht_CAN4_ADD0_Tx.Data[4]	:=	OrionBMS2_Rx.OrionBMS2_6B0_Rx.au8_Data[4];
ht_CAN4_ADD0_Tx.Data[5]	:=	OrionBMS2_Rx.OrionBMS2_6B0_Rx.au8_Data[5];		
ht_CAN4_ADD0_Tx.Data[6]	:=	OrionBMS2_Rx.OrionBMS2_6B0_Rx.au8_Data[6];	
ht_CAN4_ADD0_Tx.Data[7]	:=	OrionBMS2_Rx.OrionBMS2_6B0_Rx.au8_Data[7];		
ht_CAN4_ADD0_Tx.Len		:=	8;

ht_CAN4_ADD1_Tx.ID		:=	16#182001DD OR EPEC_CANVXD.MASK_29BIT;
ht_CAN4_ADD1_Tx.Data[0]	:=	OrionBMS2_Rx.OrionBMS2_6B1_Rx.au8_Data[0];
ht_CAN4_ADD1_Tx.Data[1]	:=	OrionBMS2_Rx.OrionBMS2_6B1_Rx.au8_Data[1];
ht_CAN4_ADD1_Tx.Data[2]	:=	OrionBMS2_Rx.OrionBMS2_6B1_Rx.au8_Data[2];
ht_CAN4_ADD1_Tx.Data[3]	:=	OrionBMS2_Rx.OrionBMS2_6B1_Rx.au8_Data[3];
ht_CAN4_ADD1_Tx.Data[4]	:=	OrionBMS2_Rx.OrionBMS2_6B1_Rx.au8_Data[4];
ht_CAN4_ADD1_Tx.Data[5]	:=	OrionBMS2_Rx.OrionBMS2_6B1_Rx.au8_Data[5];		
ht_CAN4_ADD1_Tx.Data[6]	:=	OrionBMS2_Rx.OrionBMS2_6B1_Rx.au8_Data[6];	
ht_CAN4_ADD1_Tx.Data[7]	:=	OrionBMS2_Rx.OrionBMS2_6B1_Rx.au8_Data[7];		
ht_CAN4_ADD1_Tx.Len		:=	8;

ht_CAN4_ADD2_Tx.ID		:=	16#182002DD OR EPEC_CANVXD.MASK_29BIT;
ht_CAN4_ADD2_Tx.Data[0]	:=	OrionBMS2_Rx.OrionBMS2_6B2_Rx.au8_Data[0];
ht_CAN4_ADD2_Tx.Data[1]	:=	OrionBMS2_Rx.OrionBMS2_6B2_Rx.au8_Data[1];
ht_CAN4_ADD2_Tx.Data[2]	:=	OrionBMS2_Rx.OrionBMS2_6B2_Rx.au8_Data[2];
ht_CAN4_ADD2_Tx.Data[3]	:=	OrionBMS2_Rx.OrionBMS2_6B2_Rx.au8_Data[3];
ht_CAN4_ADD2_Tx.Data[4]	:=	OrionBMS2_Rx.OrionBMS2_6B2_Rx.au8_Data[4];
ht_CAN4_ADD2_Tx.Data[5]	:=	OrionBMS2_Rx.OrionBMS2_6B2_Rx.au8_Data[5];		
ht_CAN4_ADD2_Tx.Data[6]	:=	OrionBMS2_Rx.OrionBMS2_6B2_Rx.au8_Data[6];	
ht_CAN4_ADD2_Tx.Data[7]	:=	OrionBMS2_Rx.OrionBMS2_6B2_Rx.au8_Data[7];		
ht_CAN4_ADD2_Tx.Len		:=	8;

ht_CAN4_ADD3_Tx.ID		:=	16#182003DD OR EPEC_CANVXD.MASK_29BIT;
ht_CAN4_ADD3_Tx.Data[0]	:=	OrionBMS2_Rx.OrionBMS2_6B3_Rx.au8_Data[0];
ht_CAN4_ADD3_Tx.Data[1]	:=	OrionBMS2_Rx.OrionBMS2_6B3_Rx.au8_Data[1];
ht_CAN4_ADD3_Tx.Data[2]	:=	OrionBMS2_Rx.OrionBMS2_6B3_Rx.au8_Data[2];
ht_CAN4_ADD3_Tx.Data[3]	:=	OrionBMS2_Rx.OrionBMS2_6B3_Rx.au8_Data[3];
ht_CAN4_ADD3_Tx.Data[4]	:=	OrionBMS2_Rx.OrionBMS2_6B3_Rx.au8_Data[4];
ht_CAN4_ADD3_Tx.Data[5]	:=	OrionBMS2_Rx.OrionBMS2_6B3_Rx.au8_Data[5];		
ht_CAN4_ADD3_Tx.Data[6]	:=	OrionBMS2_Rx.OrionBMS2_6B3_Rx.au8_Data[6];	
ht_CAN4_ADD3_Tx.Data[7]	:=	OrionBMS2_Rx.OrionBMS2_6B3_Rx.au8_Data[7];		
ht_CAN4_ADD3_Tx.Len		:=	8;

ht_CAN4_ADD4_Tx.ID		:=	16#182004DD OR EPEC_CANVXD.MASK_29BIT;
ht_CAN4_ADD4_Tx.Data[0]	:=	OrionBMS2_Rx.OrionBMS2_6B4_Rx.au8_Data[0];
ht_CAN4_ADD4_Tx.Data[1]	:=	OrionBMS2_Rx.OrionBMS2_6B4_Rx.au8_Data[1];
ht_CAN4_ADD4_Tx.Data[2]	:=	OrionBMS2_Rx.OrionBMS2_6B4_Rx.au8_Data[2];
ht_CAN4_ADD4_Tx.Data[3]	:=	OrionBMS2_Rx.OrionBMS2_6B4_Rx.au8_Data[3];
ht_CAN4_ADD4_Tx.Data[4]	:=	OrionBMS2_Rx.OrionBMS2_6B4_Rx.au8_Data[4];
ht_CAN4_ADD4_Tx.Data[5]	:=	OrionBMS2_Rx.OrionBMS2_6B4_Rx.au8_Data[5];		
ht_CAN4_ADD4_Tx.Data[6]	:=	OrionBMS2_Rx.OrionBMS2_6B4_Rx.au8_Data[6];	
ht_CAN4_ADD4_Tx.Data[7]	:=	OrionBMS2_Rx.OrionBMS2_6B4_Rx.au8_Data[7];		
ht_CAN4_ADD4_Tx.Len		:=	8;

ht_CAN4_ADD5_Tx.ID		:=	16#182005DD OR EPEC_CANVXD.MASK_29BIT;
ht_CAN4_ADD5_Tx.Data[0]	:=	OrionBMS2_Rx.OrionBMS2_6B5_Rx.au8_Data[0];
ht_CAN4_ADD5_Tx.Data[1]	:=	OrionBMS2_Rx.OrionBMS2_6B5_Rx.au8_Data[1];
ht_CAN4_ADD5_Tx.Data[2]	:=	OrionBMS2_Rx.OrionBMS2_6B5_Rx.au8_Data[2];
ht_CAN4_ADD5_Tx.Data[3]	:=	OrionBMS2_Rx.OrionBMS2_6B5_Rx.au8_Data[3];
ht_CAN4_ADD5_Tx.Data[4]	:=	OrionBMS2_Rx.OrionBMS2_6B5_Rx.au8_Data[4];
ht_CAN4_ADD5_Tx.Data[5]	:=	OrionBMS2_Rx.OrionBMS2_6B5_Rx.au8_Data[5];		
ht_CAN4_ADD5_Tx.Data[6]	:=	OrionBMS2_Rx.OrionBMS2_6B5_Rx.au8_Data[6];	
ht_CAN4_ADD5_Tx.Data[7]	:=	OrionBMS2_Rx.OrionBMS2_6B5_Rx.au8_Data[7];		
ht_CAN4_ADD5_Tx.Len		:=	8;

ht_CAN4_ADD6_Tx.ID		:=	16#182006DD OR EPEC_CANVXD.MASK_29BIT;
ht_CAN4_ADD6_Tx.Data[0]	:=	OrionBMS2_Rx.OrionBMS2_6B6_Rx.au8_Data[0];
ht_CAN4_ADD6_Tx.Data[1]	:=	OrionBMS2_Rx.OrionBMS2_6B6_Rx.au8_Data[1];
ht_CAN4_ADD6_Tx.Data[2]	:=	OrionBMS2_Rx.OrionBMS2_6B6_Rx.au8_Data[2];
ht_CAN4_ADD6_Tx.Data[3]	:=	OrionBMS2_Rx.OrionBMS2_6B6_Rx.au8_Data[3];
ht_CAN4_ADD6_Tx.Data[4]	:=	OrionBMS2_Rx.OrionBMS2_6B6_Rx.au8_Data[4];
ht_CAN4_ADD6_Tx.Data[5]	:=	OrionBMS2_Rx.OrionBMS2_6B6_Rx.au8_Data[5];		
ht_CAN4_ADD6_Tx.Data[6]	:=	OrionBMS2_Rx.OrionBMS2_6B6_Rx.au8_Data[6];	
ht_CAN4_ADD6_Tx.Data[7]	:=	OrionBMS2_Rx.OrionBMS2_6B6_Rx.au8_Data[7];		
ht_CAN4_ADD6_Tx.Len		:=	8;

ht_CAN4_ADD7_Tx.ID		:=	16#182007DD OR EPEC_CANVXD.MASK_29BIT;
ht_CAN4_ADD7_Tx.Data[0]	:=	OrionBMS2_Rx.OrionBMS2_6B7_Rx.au8_Data[0];
ht_CAN4_ADD7_Tx.Data[1]	:=	OrionBMS2_Rx.OrionBMS2_6B7_Rx.au8_Data[1];
ht_CAN4_ADD7_Tx.Data[2]	:=	OrionBMS2_Rx.OrionBMS2_6B7_Rx.au8_Data[2];
ht_CAN4_ADD7_Tx.Data[3]	:=	OrionBMS2_Rx.OrionBMS2_6B7_Rx.au8_Data[3];
ht_CAN4_ADD7_Tx.Data[4]	:=	OrionBMS2_Rx.OrionBMS2_6B7_Rx.au8_Data[4];
ht_CAN4_ADD7_Tx.Data[5]	:=	OrionBMS2_Rx.OrionBMS2_6B7_Rx.au8_Data[5];		
ht_CAN4_ADD7_Tx.Data[6]	:=	OrionBMS2_Rx.OrionBMS2_6B7_Rx.au8_Data[6];	
ht_CAN4_ADD7_Tx.Data[7]	:=	OrionBMS2_Rx.OrionBMS2_6B7_Rx.au8_Data[7];		
ht_CAN4_ADD7_Tx.Len		:=	8;

ht_CAN4_ADD8_Tx.ID		:=	16#182008DD OR EPEC_CANVXD.MASK_29BIT;
ht_CAN4_ADD8_Tx.Data[0]	:=	OrionBMS2_Rx.OrionBMS2_6B8_Rx.au8_Data[0];
ht_CAN4_ADD8_Tx.Data[1]	:=	OrionBMS2_Rx.OrionBMS2_6B8_Rx.au8_Data[1];
ht_CAN4_ADD8_Tx.Data[2]	:=	OrionBMS2_Rx.OrionBMS2_6B8_Rx.au8_Data[2];
ht_CAN4_ADD8_Tx.Data[3]	:=	OrionBMS2_Rx.OrionBMS2_6B8_Rx.au8_Data[3];
ht_CAN4_ADD8_Tx.Data[4]	:=	OrionBMS2_Rx.OrionBMS2_6B8_Rx.au8_Data[4];
ht_CAN4_ADD8_Tx.Data[5]	:=	OrionBMS2_Rx.OrionBMS2_6B8_Rx.au8_Data[5];		
ht_CAN4_ADD8_Tx.Data[6]	:=	OrionBMS2_Rx.OrionBMS2_6B8_Rx.au8_Data[6];	
ht_CAN4_ADD8_Tx.Data[7]	:=	OrionBMS2_Rx.OrionBMS2_6B8_Rx.au8_Data[7];		
ht_CAN4_ADD8_Tx.Len		:=	8;

ht_CAN4_ADD9_Tx.ID		:=	16#182009DD OR EPEC_CANVXD.MASK_29BIT;
ht_CAN4_ADD9_Tx.Data[0]	:=	OrionBMS2_Rx.OrionBMS2_6B9_Rx.au8_Data[0];
ht_CAN4_ADD9_Tx.Data[1]	:=	OrionBMS2_Rx.OrionBMS2_6B9_Rx.au8_Data[1];
ht_CAN4_ADD9_Tx.Data[2]	:=	OrionBMS2_Rx.OrionBMS2_6B9_Rx.au8_Data[2];
ht_CAN4_ADD9_Tx.Data[3]	:=	OrionBMS2_Rx.OrionBMS2_6B9_Rx.au8_Data[3];
ht_CAN4_ADD9_Tx.Data[4]	:=	OrionBMS2_Rx.OrionBMS2_6B9_Rx.au8_Data[4];
ht_CAN4_ADD9_Tx.Data[5]	:=	OrionBMS2_Rx.OrionBMS2_6B9_Rx.au8_Data[5];		
ht_CAN4_ADD9_Tx.Data[6]	:=	OrionBMS2_Rx.OrionBMS2_6B9_Rx.au8_Data[6];	
ht_CAN4_ADD9_Tx.Data[7]	:=	OrionBMS2_Rx.OrionBMS2_6B9_Rx.au8_Data[7];		
ht_CAN4_ADD9_Tx.Len		:=	8;

ht_CAN4_ADDA_Tx.ID		:=	16#18200ADD OR EPEC_CANVXD.MASK_29BIT;
ht_CAN4_ADDA_Tx.Data[0]	:=	OrionBMS2_Rx.OrionBMS2_6BA_Rx.au8_Data[0];
ht_CAN4_ADDA_Tx.Data[1]	:=	OrionBMS2_Rx.OrionBMS2_6BA_Rx.au8_Data[1];
ht_CAN4_ADDA_Tx.Data[2]	:=	OrionBMS2_Rx.OrionBMS2_6BA_Rx.au8_Data[2];
ht_CAN4_ADDA_Tx.Data[3]	:=	OrionBMS2_Rx.OrionBMS2_6BA_Rx.au8_Data[3];
ht_CAN4_ADDA_Tx.Data[4]	:=	OrionBMS2_Rx.OrionBMS2_6BA_Rx.au8_Data[4];
ht_CAN4_ADDA_Tx.Data[5]	:=	OrionBMS2_Rx.OrionBMS2_6BA_Rx.au8_Data[5];		
ht_CAN4_ADDA_Tx.Data[6]	:=	OrionBMS2_Rx.OrionBMS2_6BA_Rx.au8_Data[6];	
ht_CAN4_ADDA_Tx.Data[7]	:=	OrionBMS2_Rx.OrionBMS2_6BA_Rx.au8_Data[7];		
ht_CAN4_ADDA_Tx.Len		:=	8;

ht_CAN4_ADDB_Tx.ID		:=	16#18200BDD OR EPEC_CANVXD.MASK_29BIT;
ht_CAN4_ADDB_Tx.Data[0]	:=	OrionBMS2_Rx.OrionBMS2_6BB_Rx.au8_Data[0];
ht_CAN4_ADDB_Tx.Data[1]	:=	OrionBMS2_Rx.OrionBMS2_6BB_Rx.au8_Data[1];
ht_CAN4_ADDB_Tx.Data[2]	:=	OrionBMS2_Rx.OrionBMS2_6BB_Rx.au8_Data[2];
ht_CAN4_ADDB_Tx.Data[3]	:=	OrionBMS2_Rx.OrionBMS2_6BB_Rx.au8_Data[3];
ht_CAN4_ADDB_Tx.Data[4]	:=	OrionBMS2_Rx.OrionBMS2_6BB_Rx.au8_Data[4];
ht_CAN4_ADDB_Tx.Data[5]	:=	OrionBMS2_Rx.OrionBMS2_6BB_Rx.au8_Data[5];		
ht_CAN4_ADDB_Tx.Data[6]	:=	OrionBMS2_Rx.OrionBMS2_6BB_Rx.au8_Data[6];	
ht_CAN4_ADDB_Tx.Data[7]	:=	OrionBMS2_Rx.OrionBMS2_6BB_Rx.au8_Data[7];		
ht_CAN4_ADDB_Tx.Len		:=	8;

ht_CAN4_ADDC_Tx.ID		:=	16#18200CDD OR EPEC_CANVXD.MASK_29BIT;
ht_CAN4_ADDC_Tx.Data[0]	:=	OrionBMS2_Rx.OrionBMS2_6BC_Rx.au8_Data[0];
ht_CAN4_ADDC_Tx.Data[1]	:=	OrionBMS2_Rx.OrionBMS2_6BC_Rx.au8_Data[1];
ht_CAN4_ADDC_Tx.Data[2]	:=	OrionBMS2_Rx.OrionBMS2_6BC_Rx.au8_Data[2];
ht_CAN4_ADDC_Tx.Data[3]	:=	OrionBMS2_Rx.OrionBMS2_6BC_Rx.au8_Data[3];
ht_CAN4_ADDC_Tx.Data[4]	:=	OrionBMS2_Rx.OrionBMS2_6BC_Rx.au8_Data[4];
ht_CAN4_ADDC_Tx.Data[5]	:=	OrionBMS2_Rx.OrionBMS2_6BC_Rx.au8_Data[5];		
ht_CAN4_ADDC_Tx.Data[6]	:=	OrionBMS2_Rx.OrionBMS2_6BC_Rx.au8_Data[6];	
ht_CAN4_ADDC_Tx.Data[7]	:=	OrionBMS2_Rx.OrionBMS2_6BC_Rx.au8_Data[7];		
ht_CAN4_ADDC_Tx.Len		:=	8;

ht_CAN4_ADDD_Tx.ID		:=	16#18200DDD OR EPEC_CANVXD.MASK_29BIT;
ht_CAN4_ADDD_Tx.Data[0]	:=	OrionBMS2_Rx.OrionBMS2_6BD_Rx.au8_Data[0];
ht_CAN4_ADDD_Tx.Data[1]	:=	OrionBMS2_Rx.OrionBMS2_6BD_Rx.au8_Data[1];
ht_CAN4_ADDD_Tx.Data[2]	:=	OrionBMS2_Rx.OrionBMS2_6BD_Rx.au8_Data[2];
ht_CAN4_ADDD_Tx.Data[3]	:=	OrionBMS2_Rx.OrionBMS2_6BD_Rx.au8_Data[3];
ht_CAN4_ADDD_Tx.Data[4]	:=	OrionBMS2_Rx.OrionBMS2_6BD_Rx.au8_Data[4];
ht_CAN4_ADDD_Tx.Data[5]	:=	OrionBMS2_Rx.OrionBMS2_6BD_Rx.au8_Data[5];		
ht_CAN4_ADDD_Tx.Data[6]	:=	OrionBMS2_Rx.OrionBMS2_6BD_Rx.au8_Data[6];	
ht_CAN4_ADDD_Tx.Data[7]	:=	OrionBMS2_Rx.OrionBMS2_6BD_Rx.au8_Data[7];		
ht_CAN4_ADDD_Tx.Len		:=	8;



Tx_Timer(IN := NOT(Tx_Timer.Q), PT := T#1000MS);
IF (Tx_Timer.Q = TRUE) THEN
	G_CAN4_Channel.SendMessage(i_pMSG:=ADR(ht_CAN4_DD0_Tx));
	G_CAN4_Channel.SendMessage(i_pMSG:=ADR(ht_CAN4_DD1_Tx));
	G_CAN4_Channel.SendMessage(i_pMSG:=ADR(ht_CAN4_DD2_Tx));
	G_CAN4_Channel.SendMessage(i_pMSG:=ADR(ht_CAN4_DD3_Tx));
	G_CAN4_Channel.SendMessage(i_pMSG:=ADR(ht_CAN4_DD4_Tx));
	G_CAN4_Channel.SendMessage(i_pMSG:=ADR(ht_CAN4_DD5_Tx));
	G_CAN4_Channel.SendMessage(i_pMSG:=ADR(ht_CAN4_DD6_Tx));
	G_CAN4_Channel.SendMessage(i_pMSG:=ADR(ht_CAN4_DD7_Tx));
	G_CAN4_Channel.SendMessage(i_pMSG:=ADR(ht_CAN4_DD8_Tx));
	G_CAN4_Channel.SendMessage(i_pMSG:=ADR(ht_CAN4_DD9_Tx));
	G_CAN4_Channel.SendMessage(i_pMSG:=ADR(ht_CAN4_DDA_Tx));
	G_CAN4_Channel.SendMessage(i_pMSG:=ADR(ht_CAN4_DDB_Tx));
	G_CAN4_Channel.SendMessage(i_pMSG:=ADR(ht_CAN4_DDC_Tx));
	G_CAN4_Channel.SendMessage(i_pMSG:=ADR(ht_CAN4_DDD_Tx));
	G_CAN4_Channel.SendMessage(i_pMSG:=ADR(ht_CAN4_ADD0_Tx));
	G_CAN4_Channel.SendMessage(i_pMSG:=ADR(ht_CAN4_ADD1_Tx));
	G_CAN4_Channel.SendMessage(i_pMSG:=ADR(ht_CAN4_ADD2_Tx));
	G_CAN4_Channel.SendMessage(i_pMSG:=ADR(ht_CAN4_ADD3_Tx));
	G_CAN4_Channel.SendMessage(i_pMSG:=ADR(ht_CAN4_ADD4_Tx));
	G_CAN4_Channel.SendMessage(i_pMSG:=ADR(ht_CAN4_ADD5_Tx));
	G_CAN4_Channel.SendMessage(i_pMSG:=ADR(ht_CAN4_ADD6_Tx));
	G_CAN4_Channel.SendMessage(i_pMSG:=ADR(ht_CAN4_ADD7_Tx));
	G_CAN4_Channel.SendMessage(i_pMSG:=ADR(ht_CAN4_ADD8_Tx));
	G_CAN4_Channel.SendMessage(i_pMSG:=ADR(ht_CAN4_ADD9_Tx));
	G_CAN4_Channel.SendMessage(i_pMSG:=ADR(ht_CAN4_ADDA_Tx));
	G_CAN4_Channel.SendMessage(i_pMSG:=ADR(ht_CAN4_ADDB_Tx));
	G_CAN4_Channel.SendMessage(i_pMSG:=ADR(ht_CAN4_ADDC_Tx));
	G_CAN4_Channel.SendMessage(i_pMSG:=ADR(ht_CAN4_ADDD_Tx));
	
END_IF

END_PROGRAM

// Application/UserCode/HMI/Data to or For HMI/BRUSA_to_HMI_1
PROGRAM BRUSA_to_HMI_1
VAR
	ht_CAN4_7DD0_Tx	:	EPEC_CANVXD.Msg;
	ht_CAN4_7DD1_Tx	:	EPEC_CANVXD.Msg;
	ht_CAN4_7DD2_Tx: EPEC_CANVXD.msg;
	ht_CAN4_7DD3_Tx: EPEC_CANVXD.msg;
	ht_CAN4_7DD4_Tx: EPEC_CANVXD.msg;
	ht_CAN4_7DD5_Tx: EPEC_CANVXD.msg;
	ht_CAN4_7DD6_Tx: EPEC_CANVXD.msg;
	ht_CAN4_7DD7_Tx: EPEC_CANVXD.msg;
	ht_CAN4_7DD8_Tx: EPEC_CANVXD.msg;
	ht_CAN4_7DD9_Tx: EPEC_CANVXD.msg;
	ht_CAN4_7DDA_Tx: EPEC_CANVXD.msg;
	ht_CAN4_7DDB_Tx: EPEC_CANVXD.msg;
	hton_MessageSend_Timer	:	TON;
	Tx_Timer	:	TON;
	END_VAR

//called from can4_TX

//Master Brusa
ht_CAN4_7DD0_Tx.ID		:=	16#187000DD OR EPEC_CANVXD.MASK_29BIT;
ht_CAN4_7DD0_Tx.Data[0]	:=	Brusa1_Rx.ActAC_Rx.au8_Data[0];
ht_CAN4_7DD0_Tx.Data[1]	:=	Brusa1_Rx.ActAC_Rx.au8_Data[1];
ht_CAN4_7DD0_Tx.Data[2]	:=	Brusa1_Rx.ActAC_Rx.au8_Data[2];
ht_CAN4_7DD0_Tx.Data[3]	:=	Brusa1_Rx.ActAC_Rx.au8_Data[3];
ht_CAN4_7DD0_Tx.Data[4]	:=	Brusa1_Rx.ActAC_Rx.au8_Data[4];
ht_CAN4_7DD0_Tx.Data[5]	:=	Brusa1_Rx.ActAC_Rx.au8_Data[5];
ht_CAN4_7DD0_Tx.Data[6]	:=	Brusa1_Rx.ActAC_Rx.au8_Data[6];
ht_CAN4_7DD0_Tx.Data[7]	:=	Brusa1_Rx.ActAC_Rx.au8_Data[7];
ht_CAN4_7DD0_Tx.Len		:=	8;

//* Errors
ht_CAN4_7DD2_Tx.ID		:=	16#187002DD OR EPEC_CANVXD.MASK_29BIT;
ht_CAN4_7DD2_Tx.Data[0]	:=	Brusa1_Rx.ActErr_Rx.au8_Data[0];
ht_CAN4_7DD2_Tx.Data[1]	:=	Brusa1_Rx.ActErr_Rx.au8_Data[1];
ht_CAN4_7DD2_Tx.Data[2]	:=	Brusa1_Rx.ActErr_Rx.au8_Data[2];
ht_CAN4_7DD2_Tx.Data[3]	:=	Brusa1_Rx.ActErr_Rx.au8_Data[3];
ht_CAN4_7DD2_Tx.Data[4]	:=	Brusa1_Rx.ActErr_Rx.au8_Data[4];
ht_CAN4_7DD2_Tx.Data[5]	:=	Brusa1_Rx.ActErr_Rx.au8_Data[5];
ht_CAN4_7DD2_Tx.Data[6]	:=	Brusa1_Rx.ActErr_Rx.au8_Data[6];
ht_CAN4_7DD2_Tx.Data[7]	:=	Brusa1_Rx.ActErr_Rx.au8_Data[7];
ht_CAN4_7DD2_Tx.Len		:=	8;

ht_CAN4_7DD4_Tx.ID		:=	16#187004DD OR EPEC_CANVXD.MASK_29BIT;
ht_CAN4_7DD4_Tx.Data[0]	:=	Brusa1_Rx.ActInt_Rx.au8_Data[0];
ht_CAN4_7DD4_Tx.Data[1]	:=	Brusa1_Rx.ActInt_Rx.au8_Data[1];
ht_CAN4_7DD4_Tx.Data[2]	:=	Brusa1_Rx.ActInt_Rx.au8_Data[2];
ht_CAN4_7DD4_Tx.Data[3]	:=	Brusa1_Rx.ActInt_Rx.au8_Data[3];
ht_CAN4_7DD4_Tx.Data[4]	:=	Brusa1_Rx.ActInt_Rx.au8_Data[4];
ht_CAN4_7DD4_Tx.Data[5]	:=	Brusa1_Rx.ActInt_Rx.au8_Data[5];
ht_CAN4_7DD4_Tx.Data[6]	:=	Brusa1_Rx.ActInt_Rx.au8_Data[6];
ht_CAN4_7DD4_Tx.Data[7]	:=	Brusa1_Rx.ActInt_Rx.au8_Data[7];
ht_CAN4_7DD4_Tx.Len		:=	8;

ht_CAN4_7DD6_Tx.ID		:=	16#187006DD OR EPEC_CANVXD.MASK_29BIT;
ht_CAN4_7DD6_Tx.Data[0]	:=	Brusa1_Rx.ActLim_Rx.au8_Data[0];
ht_CAN4_7DD6_Tx.Data[1]	:=	Brusa1_Rx.ActLim_Rx.au8_Data[1];
ht_CAN4_7DD6_Tx.Data[2]	:=	Brusa1_Rx.ActLim_Rx.au8_Data[2];
ht_CAN4_7DD6_Tx.Data[3]	:=	Brusa1_Rx.ActLim_Rx.au8_Data[3];
ht_CAN4_7DD6_Tx.Data[4]	:=	Brusa1_Rx.ActLim_Rx.au8_Data[4];
ht_CAN4_7DD6_Tx.Data[5]	:=	Brusa1_Rx.ActLim_Rx.au8_Data[5];
ht_CAN4_7DD6_Tx.Data[6]	:=	Brusa1_Rx.ActLim_Rx.au8_Data[6];
ht_CAN4_7DD6_Tx.Data[7]	:=	Brusa1_Rx.ActLim_Rx.au8_Data[7];
ht_CAN4_7DD6_Tx.Len		:=	8;

ht_CAN4_7DD8_Tx.ID		:=	16#187008DD OR EPEC_CANVXD.MASK_29BIT;
ht_CAN4_7DD8_Tx.Data[0]	:=	Brusa1_Rx.ActPlug_Rx.au8_Data[0];
ht_CAN4_7DD8_Tx.Data[1]	:=	Brusa1_Rx.ActPlug_Rx.au8_Data[1];
ht_CAN4_7DD8_Tx.Data[2]	:=	Brusa1_Rx.ActPlug_Rx.au8_Data[2];
ht_CAN4_7DD8_Tx.Data[3]	:=	Brusa1_Rx.ActPlug_Rx.au8_Data[3];
ht_CAN4_7DD8_Tx.Data[4]	:=	Brusa1_Rx.ActPlug_Rx.au8_Data[4];
ht_CAN4_7DD8_Tx.Data[5]	:=	Brusa1_Rx.ActPlug_Rx.au8_Data[5];
ht_CAN4_7DD8_Tx.Data[6]	:=	Brusa1_Rx.ActPlug_Rx.au8_Data[6];
ht_CAN4_7DD8_Tx.Data[7]	:=	Brusa1_Rx.ActPlug_Rx.au8_Data[7];
ht_CAN4_7DD8_Tx.Len		:=	8;

ht_CAN4_7DDA_Tx.ID		:=	16#18700ADD OR EPEC_CANVXD.MASK_29BIT;
ht_CAN4_7DDA_Tx.Data[0]	:=	Brusa1_Tx.DenLim_Tx.Data[0];
ht_CAN4_7DDA_Tx.Data[1]	:=	Brusa1_Tx.DenLim_Tx.Data[1];
ht_CAN4_7DDA_Tx.Data[2]	:=	Brusa1_Tx.DenLim_Tx.Data[2];
ht_CAN4_7DDA_Tx.Data[3]	:=	Brusa1_Tx.DenLim_Tx.Data[3];
ht_CAN4_7DDA_Tx.Data[4]	:=	Brusa1_Tx.DenLim_Tx.Data[4];
ht_CAN4_7DDA_Tx.Data[5]	:=	Brusa1_Tx.DenLim_Tx.Data[5];
ht_CAN4_7DDA_Tx.Data[6]	:=	Brusa1_Tx.DenLim_Tx.Data[6];
ht_CAN4_7DDA_Tx.Data[7]	:=	Brusa1_Tx.DenLim_Tx.Data[7];
ht_CAN4_7DDA_Tx.Len		:=	8;



//Slave Brusa
ht_CAN4_7DD1_Tx.ID		:=	16#187001DD OR EPEC_CANVXD.MASK_29BIT;
ht_CAN4_7DD1_Tx.Data[0]	:=	Brusa2_Rx.ActAC_Rx.au8_Data[0];
ht_CAN4_7DD1_Tx.Data[1]	:=	Brusa2_Rx.ActAC_Rx.au8_Data[1];
ht_CAN4_7DD1_Tx.Data[2]	:=	Brusa2_Rx.ActAC_Rx.au8_Data[2];
ht_CAN4_7DD1_Tx.Data[3]	:=	Brusa2_Rx.ActAC_Rx.au8_Data[3];
ht_CAN4_7DD1_Tx.Data[4]	:=	Brusa2_Rx.ActAC_Rx.au8_Data[4];
ht_CAN4_7DD1_Tx.Data[5]	:=	Brusa2_Rx.ActAC_Rx.au8_Data[5];
ht_CAN4_7DD1_Tx.Data[6]	:=	Brusa2_Rx.ActAC_Rx.au8_Data[6];
ht_CAN4_7DD1_Tx.Data[7]	:=	Brusa2_Rx.ActAC_Rx.au8_Data[7];
ht_CAN4_7DD1_Tx.Len		:=	8;

ht_CAN4_7DD3_Tx.ID		:=	16#187003DD OR EPEC_CANVXD.MASK_29BIT;
ht_CAN4_7DD3_Tx.Data[0]	:=	Brusa2_Rx.NLG2_ActErr_Rx.au8_Data[0];
ht_CAN4_7DD3_Tx.Data[1]	:=	Brusa2_Rx.NLG2_ActErr_Rx.au8_Data[1];
ht_CAN4_7DD3_Tx.Data[2]	:=	Brusa2_Rx.NLG2_ActErr_Rx.au8_Data[2];
ht_CAN4_7DD3_Tx.Data[3]	:=	Brusa2_Rx.NLG2_ActErr_Rx.au8_Data[3];
ht_CAN4_7DD3_Tx.Data[4]	:=	Brusa2_Rx.NLG2_ActErr_Rx.au8_Data[4];
ht_CAN4_7DD3_Tx.Data[5]	:=	Brusa2_Rx.NLG2_ActErr_Rx.au8_Data[5];
ht_CAN4_7DD3_Tx.Data[6]	:=	Brusa2_Rx.NLG2_ActErr_Rx.au8_Data[6];
ht_CAN4_7DD3_Tx.Data[7]	:=	Brusa2_Rx.NLG2_ActErr_Rx.au8_Data[7];
ht_CAN4_7DD3_Tx.Len		:=	8;

ht_CAN4_7DD5_Tx.ID		:=	16#187005DD OR EPEC_CANVXD.MASK_29BIT;
ht_CAN4_7DD5_Tx.Data[0]	:=	Brusa2_Rx.NLG2_ActInt_Rx.au8_Data[0];
ht_CAN4_7DD5_Tx.Data[1]	:=	Brusa2_Rx.NLG2_ActInt_Rx.au8_Data[1];
ht_CAN4_7DD5_Tx.Data[2]	:=	Brusa2_Rx.NLG2_ActInt_Rx.au8_Data[2];
ht_CAN4_7DD5_Tx.Data[3]	:=	Brusa2_Rx.NLG2_ActInt_Rx.au8_Data[3];
ht_CAN4_7DD5_Tx.Data[4]	:=	Brusa2_Rx.NLG2_ActInt_Rx.au8_Data[4];
ht_CAN4_7DD5_Tx.Data[5]	:=	Brusa2_Rx.NLG2_ActInt_Rx.au8_Data[5];
ht_CAN4_7DD5_Tx.Data[6]	:=	Brusa2_Rx.NLG2_ActInt_Rx.au8_Data[6];
ht_CAN4_7DD5_Tx.Data[7]	:=	Brusa2_Rx.NLG2_ActInt_Rx.au8_Data[7];
ht_CAN4_7DD5_Tx.Len		:=	8;

ht_CAN4_7DD7_Tx.ID		:=	16#187007DD OR EPEC_CANVXD.MASK_29BIT;
ht_CAN4_7DD7_Tx.Data[0]	:=	Brusa2_Rx.NLG2_ActLim_Rx.au8_Data[0];
ht_CAN4_7DD7_Tx.Data[1]	:=	Brusa2_Rx.NLG2_ActLim_Rx.au8_Data[1];
ht_CAN4_7DD7_Tx.Data[2]	:=	Brusa2_Rx.NLG2_ActLim_Rx.au8_Data[2];
ht_CAN4_7DD7_Tx.Data[3]	:=	Brusa2_Rx.NLG2_ActLim_Rx.au8_Data[3];
ht_CAN4_7DD7_Tx.Data[4]	:=	Brusa2_Rx.NLG2_ActLim_Rx.au8_Data[4];
ht_CAN4_7DD7_Tx.Data[5]	:=	Brusa2_Rx.NLG2_ActLim_Rx.au8_Data[5];
ht_CAN4_7DD7_Tx.Data[6]	:=	Brusa2_Rx.NLG2_ActLim_Rx.au8_Data[6];
ht_CAN4_7DD7_Tx.Data[7]	:=	Brusa2_Rx.NLG2_ActLim_Rx.au8_Data[7];
ht_CAN4_7DD7_Tx.Len		:=	8;

ht_CAN4_7DD9_Tx.ID		:=	16#187009DD OR EPEC_CANVXD.MASK_29BIT;
ht_CAN4_7DD9_Tx.Data[0]	:=	Brusa2_Rx.NLG2_ActPlug_Rx.au8_Data[0];
ht_CAN4_7DD9_Tx.Data[1]	:=	Brusa2_Rx.NLG2_ActPlug_Rx.au8_Data[1];
ht_CAN4_7DD9_Tx.Data[2]	:=	Brusa2_Rx.NLG2_ActPlug_Rx.au8_Data[2];
ht_CAN4_7DD9_Tx.Data[3]	:=	Brusa2_Rx.NLG2_ActPlug_Rx.au8_Data[3];
ht_CAN4_7DD9_Tx.Data[4]	:=	Brusa2_Rx.NLG2_ActPlug_Rx.au8_Data[4];
ht_CAN4_7DD9_Tx.Data[5]	:=	Brusa2_Rx.NLG2_ActPlug_Rx.au8_Data[5];
ht_CAN4_7DD9_Tx.Data[6]	:=	Brusa2_Rx.NLG2_ActPlug_Rx.au8_Data[6];
ht_CAN4_7DD9_Tx.Data[7]	:=	Brusa2_Rx.NLG2_ActPlug_Rx.au8_Data[7];
ht_CAN4_7DD9_Tx.Len		:=	8;

ht_CAN4_7DDB_Tx.ID		:=	16#18700BDD OR EPEC_CANVXD.MASK_29BIT;
ht_CAN4_7DDB_Tx.Data[0]	:=	Brusa2_Tx.DenLim_Tx.Data[0];
ht_CAN4_7DDB_Tx.Data[1]	:=	Brusa2_Tx.DenLim_Tx.Data[1];
ht_CAN4_7DDB_Tx.Data[2]	:=	Brusa2_Tx.DenLim_Tx.Data[2];
ht_CAN4_7DDB_Tx.Data[3]	:=	Brusa2_Tx.DenLim_Tx.Data[3];
ht_CAN4_7DDB_Tx.Data[4]	:=	Brusa2_Tx.DenLim_Tx.Data[4];
ht_CAN4_7DDB_Tx.Data[5]	:=	Brusa2_Tx.DenLim_Tx.Data[5];
ht_CAN4_7DDB_Tx.Data[6]	:=	Brusa2_Tx.DenLim_Tx.Data[6];
ht_CAN4_7DDB_Tx.Data[7]	:=	Brusa2_Tx.DenLim_Tx.Data[7];
ht_CAN4_7DDB_Tx.Len		:=	8;



Tx_Timer(IN := NOT(Tx_Timer.Q), PT := T#100MS);
IF (Tx_Timer.Q = TRUE) THEN
	G_CAN4_Channel.SendMessage(i_pMSG:=ADR(ht_CAN4_7DD0_Tx));
	G_CAN4_Channel.SendMessage(i_pMSG:=ADR(ht_CAN4_7DD1_Tx));
	G_CAN4_Channel.SendMessage(i_pMSG:=ADR(ht_CAN4_7DD2_Tx));
	G_CAN4_Channel.SendMessage(i_pMSG:=ADR(ht_CAN4_7DD3_Tx));
	G_CAN4_Channel.SendMessage(i_pMSG:=ADR(ht_CAN4_7DD4_Tx));
	G_CAN4_Channel.SendMessage(i_pMSG:=ADR(ht_CAN4_7DD5_Tx));
	G_CAN4_Channel.SendMessage(i_pMSG:=ADR(ht_CAN4_7DD6_Tx));
	G_CAN4_Channel.SendMessage(i_pMSG:=ADR(ht_CAN4_7DD7_Tx));
	G_CAN4_Channel.SendMessage(i_pMSG:=ADR(ht_CAN4_7DD8_Tx));
	G_CAN4_Channel.SendMessage(i_pMSG:=ADR(ht_CAN4_7DD9_Tx));
	G_CAN4_Channel.SendMessage(i_pMSG:=ADR(ht_CAN4_7DDA_Tx));
	G_CAN4_Channel.SendMessage(i_pMSG:=ADR(ht_CAN4_7DDB_Tx));
END_IF

END_PROGRAM

// Application/UserCode/HMI/Data to or For HMI/DCDC_to_HMI_1
PROGRAM DCDC_to_HMI_1
VAR
	ht_CAN4_5DD0_Tx	:	EPEC_CANVXD.Msg;
	ht_CAN4_5DD1_Tx: 	EPEC_CANVXD.Msg;
	hton_MessageSend_Timer	:	TON;
	
	Tx_Timer	:	TON;
	
END_VAR


//DCDC
ht_CAN4_5DD0_Tx.ID		:=	16#185000DD OR EPEC_CANVXD.MASK_29BIT;
ht_CAN4_5DD0_Tx.Data[0]	:=	BELDCDC_Rx.BelDCDC_IO_Rx.au8_Data[0];
ht_CAN4_5DD0_Tx.Data[1]	:=	BELDCDC_Rx.BelDCDC_IO_Rx.au8_Data[1];
ht_CAN4_5DD0_Tx.Data[2]	:=	BELDCDC_Rx.BelDCDC_IO_Rx.au8_Data[2];
ht_CAN4_5DD0_Tx.Data[3]	:=	BELDCDC_Rx.BelDCDC_IO_Rx.au8_Data[3];
ht_CAN4_5DD0_Tx.Data[4]	:=	BELDCDC_Rx.BelDCDC_IO_Rx.au8_Data[4];
ht_CAN4_5DD0_Tx.Data[5]	:=	BELDCDC_Rx.BelDCDC_IO_Rx.au8_Data[5];	
ht_CAN4_5DD0_Tx.Data[6]	:=	BELDCDC_Rx.BelDCDC_IO_Rx.au8_Data[6];	
ht_CAN4_5DD0_Tx.Data[7]	:=	BELDCDC_Rx.BelDCDC_IO_Rx.au8_Data[7];	
ht_CAN4_5DD0_Tx.Len		:=	8;

ht_CAN4_5DD1_Tx.ID		:=	16#185001DD OR EPEC_CANVXD.MASK_29BIT;
ht_CAN4_5DD1_Tx.Data[0]	:=	BELDCDC_Rx.BelDCDC_FWS_Rx.au8_Data[0];
ht_CAN4_5DD1_Tx.Data[1]	:=	BELDCDC_Rx.BelDCDC_FWS_Rx.au8_Data[1];
ht_CAN4_5DD1_Tx.Data[2]	:=	BELDCDC_Rx.BelDCDC_FWS_Rx.au8_Data[2];
ht_CAN4_5DD1_Tx.Data[3]	:=	BELDCDC_Rx.BelDCDC_FWS_Rx.au8_Data[3];
ht_CAN4_5DD1_Tx.Data[4]	:=	BELDCDC_Rx.BelDCDC_FWS_Rx.au8_Data[4];
ht_CAN4_5DD1_Tx.Data[5]	:=	BELDCDC_Rx.BelDCDC_FWS_Rx.au8_Data[5];	
ht_CAN4_5DD1_Tx.Data[6]	:=	BELDCDC_Rx.BelDCDC_FWS_Rx.au8_Data[6];	
ht_CAN4_5DD1_Tx.Data[7]	:=	BELDCDC_Rx.BelDCDC_FWS_Rx.au8_Data[7];	
ht_CAN4_5DD1_Tx.Len		:=	8;


Tx_Timer(IN := NOT(Tx_Timer.Q), PT := T#1000MS);
IF (Tx_Timer.Q = TRUE) THEN
	G_CAN4_Channel.SendMessage(i_pMSG:=ADR(ht_CAN4_5DD0_Tx));
	G_CAN4_Channel.SendMessage(i_pMSG:=ADR(ht_CAN4_5DD1_Tx));
	
	END_IF

END_PROGRAM

// Application/UserCode/HMI/Data to or For HMI/MCU_to_HMI_1
PROGRAM MCU_to_HMI_1
VAR
	ht_CAN4_6DD0_Tx	:	EPEC_CANVXD.Msg;
	ht_CAN4_6DD1_Tx	:	EPEC_CANVXD.Msg;
	ht_CAN4_6DD2_Tx	:	EPEC_CANVXD.Msg;
	ht_CAN4_6DD3_Tx: EPEC_CANVXD.Msg;
	ht_CAN4_6DD4_Tx: EPEC_CANVXD.Msg;
	ht_CAN4_6DD5_Tx: EPEC_CANVXD.Msg;
	ht_CAN4_6DD6_Tx: EPEC_CANVXD.Msg;
	ht_CAN4_6DD7_Tx: EPEC_CANVXD.Msg;
	ht_CAN4_6DD8_Tx: EPEC_CANVXD.Msg;
	hton_MessageSend_Timer	:	TON;
	
	Tx_Timer	:	TON;
	
END_VAR


//MCU
ht_CAN4_6DD0_Tx.ID		:=	16#186000DD OR EPEC_CANVXD.MASK_29BIT;
ht_CAN4_6DD0_Tx.Data[0]	:=	MCU_Rx.MCU_Info1_Rx.au8_Data[0];
ht_CAN4_6DD0_Tx.Data[1]	:=	MCU_Rx.MCU_Info1_Rx.au8_Data[1];
ht_CAN4_6DD0_Tx.Data[2]	:=	MCU_Rx.MCU_Info1_Rx.au8_Data[2];
ht_CAN4_6DD0_Tx.Data[3]	:=	MCU_Rx.MCU_Info1_Rx.au8_Data[3];
ht_CAN4_6DD0_Tx.Data[4]	:=	MCU_Rx.MCU_Info1_Rx.au8_Data[4];
ht_CAN4_6DD0_Tx.Data[5]	:=	MCU_Rx.MCU_Info1_Rx.au8_Data[5];
ht_CAN4_6DD0_Tx.Data[6]	:=	MCU_Rx.MCU_Info1_Rx.au8_Data[6];
ht_CAN4_6DD0_Tx.Data[7]	:=	MCU_Rx.MCU_Info1_Rx.au8_Data[7];
ht_CAN4_6DD0_Tx.Len		:=	8;

ht_CAN4_6DD1_Tx.ID		:=	16#186001DD OR EPEC_CANVXD.MASK_29BIT;
ht_CAN4_6DD1_Tx.Data[0]	:=	MCU_Rx.MCU_Info2_Rx.au8_Data[0];
ht_CAN4_6DD1_Tx.Data[1]	:=	MCU_Rx.MCU_Info2_Rx.au8_Data[1];
ht_CAN4_6DD1_Tx.Data[2]	:=	MCU_Rx.MCU_Info2_Rx.au8_Data[2];
ht_CAN4_6DD1_Tx.Data[3]	:=	MCU_Rx.MCU_Info2_Rx.au8_Data[3];
ht_CAN4_6DD1_Tx.Data[4]	:=	MCU_Rx.MCU_Info2_Rx.au8_Data[4];
ht_CAN4_6DD1_Tx.Data[5]	:=	MCU_Rx.MCU_Info2_Rx.au8_Data[5];
ht_CAN4_6DD1_Tx.Data[6]	:=	MCU_Rx.MCU_Info2_Rx.au8_Data[6];
ht_CAN4_6DD1_Tx.Data[7]	:=	MCU_Rx.MCU_Info2_Rx.au8_Data[7];
ht_CAN4_6DD1_Tx.Len		:=	8;

ht_CAN4_6DD2_Tx.ID		:=	16#186002DD OR EPEC_CANVXD.MASK_29BIT;
ht_CAN4_6DD2_Tx.Data[0]	:=	MCU_Tx.ht_MCU_VMUComm1_Tx.Data[0];
ht_CAN4_6DD2_Tx.Data[1]	:=	MCU_Tx.ht_MCU_VMUComm1_Tx.Data[1];
ht_CAN4_6DD2_Tx.Data[2]	:=	MCU_Tx.ht_MCU_VMUComm1_Tx.Data[2];
ht_CAN4_6DD2_Tx.Data[3]	:=	MCU_Tx.ht_MCU_VMUComm1_Tx.Data[3];
ht_CAN4_6DD2_Tx.Data[4]	:=	MCU_Tx.ht_MCU_VMUComm1_Tx.Data[4];
ht_CAN4_6DD2_Tx.Data[5]	:=	MCU_Tx.ht_MCU_VMUComm1_Tx.Data[5];
ht_CAN4_6DD2_Tx.Data[6]	:=	MCU_Tx.ht_MCU_VMUComm1_Tx.Data[6];
ht_CAN4_6DD2_Tx.Data[7]	:=	MCU_Tx.ht_MCU_VMUComm1_Tx.Data[7];
ht_CAN4_6DD2_Tx.Len		:=	8;

ht_CAN4_6DD3_Tx.ID		:=	16#186003DD OR EPEC_CANVXD.MASK_29BIT;
ht_CAN4_6DD3_Tx.Data[0]	:=	MCU_Tx.ht_MCU_VMUComm2_Tx.Data[0];
ht_CAN4_6DD3_Tx.Data[1]	:=	MCU_Tx.ht_MCU_VMUComm2_Tx.Data[1];
ht_CAN4_6DD3_Tx.Data[2]	:=	MCU_Tx.ht_MCU_VMUComm2_Tx.Data[2];
ht_CAN4_6DD3_Tx.Data[3]	:=	MCU_Tx.ht_MCU_VMUComm2_Tx.Data[3];
ht_CAN4_6DD3_Tx.Data[4]	:=	MCU_Tx.ht_MCU_VMUComm2_Tx.Data[4];
ht_CAN4_6DD3_Tx.Data[5]	:=	MCU_Tx.ht_MCU_VMUComm2_Tx.Data[5];
ht_CAN4_6DD3_Tx.Data[6]	:=	MCU_Tx.ht_MCU_VMUComm2_Tx.Data[6];
ht_CAN4_6DD3_Tx.Data[7]	:=	MCU_Tx.ht_MCU_VMUComm2_Tx.Data[7];
ht_CAN4_6DD3_Tx.Len		:=	8;

ht_CAN4_6DD5_Tx.ID		:=	16#186005DD OR EPEC_CANVXD.MASK_29BIT;
ht_CAN4_6DD5_Tx.Data[0]	:=	MCU_Rx.MCU_CommandResponse1_Rx.au8_Data[0];
ht_CAN4_6DD5_Tx.Data[1]	:=	MCU_Rx.MCU_CommandResponse1_Rx.au8_Data[1];
ht_CAN4_6DD5_Tx.Data[2]	:=	MCU_Rx.MCU_CommandResponse1_Rx.au8_Data[2];
ht_CAN4_6DD5_Tx.Data[3]	:=	MCU_Rx.MCU_CommandResponse1_Rx.au8_Data[3];
ht_CAN4_6DD5_Tx.Data[4]	:=	MCU_Rx.MCU_CommandResponse1_Rx.au8_Data[4];
ht_CAN4_6DD5_Tx.Data[5]	:=	MCU_Rx.MCU_CommandResponse1_Rx.au8_Data[5];
ht_CAN4_6DD5_Tx.Data[6]	:=	MCU_Rx.MCU_CommandResponse1_Rx.au8_Data[6];
ht_CAN4_6DD5_Tx.Data[7]	:=	MCU_Rx.MCU_CommandResponse1_Rx.au8_Data[7];
ht_CAN4_6DD5_Tx.Len		:=	8;

ht_CAN4_6DD6_Tx.ID		:=	16#186006DD OR EPEC_CANVXD.MASK_29BIT;
ht_CAN4_6DD6_Tx.Data[0]	:=	MCU_Rx.MCU_CommandResponse2_Rx.au8_Data[0];
ht_CAN4_6DD6_Tx.Data[1]	:=	MCU_Rx.MCU_CommandResponse2_Rx.au8_Data[1];
ht_CAN4_6DD6_Tx.Data[2]	:=	MCU_Rx.MCU_CommandResponse2_Rx.au8_Data[2];
ht_CAN4_6DD6_Tx.Data[3]	:=	MCU_Rx.MCU_CommandResponse2_Rx.au8_Data[3];
ht_CAN4_6DD6_Tx.Data[4]	:=	MCU_Rx.MCU_CommandResponse2_Rx.au8_Data[4];
ht_CAN4_6DD6_Tx.Data[5]	:=	MCU_Rx.MCU_CommandResponse2_Rx.au8_Data[5];
ht_CAN4_6DD6_Tx.Data[6]	:=	MCU_Rx.MCU_CommandResponse2_Rx.au8_Data[6];
ht_CAN4_6DD6_Tx.Data[7]	:=	MCU_Rx.MCU_CommandResponse2_Rx.au8_Data[7];
ht_CAN4_6DD6_Tx.Len		:=	8;

ht_CAN4_6DD7_Tx.ID		:=	16#186007DD OR EPEC_CANVXD.MASK_29BIT;
ht_CAN4_6DD7_Tx.Data[0]	:=	MCU_Rx.MCU_EventInfo1_Rx.au8_Data[0];
ht_CAN4_6DD7_Tx.Data[1]	:=	MCU_Rx.MCU_EventInfo1_Rx.au8_Data[1];
ht_CAN4_6DD7_Tx.Data[2]	:=	MCU_Rx.MCU_EventInfo1_Rx.au8_Data[2];
ht_CAN4_6DD7_Tx.Data[3]	:=	MCU_Rx.MCU_EventInfo1_Rx.au8_Data[3];
ht_CAN4_6DD7_Tx.Data[4]	:=	MCU_Rx.MCU_EventInfo1_Rx.au8_Data[4];
ht_CAN4_6DD7_Tx.Data[5]	:=	MCU_Rx.MCU_EventInfo1_Rx.au8_Data[5];
ht_CAN4_6DD7_Tx.Data[6]	:=	MCU_Rx.MCU_EventInfo1_Rx.au8_Data[6];
ht_CAN4_6DD7_Tx.Data[7]	:=	MCU_Rx.MCU_EventInfo1_Rx.au8_Data[7];
ht_CAN4_6DD7_Tx.Len		:=	8;

ht_CAN4_6DD8_Tx.ID		:=	16#186008DD OR EPEC_CANVXD.MASK_29BIT;
ht_CAN4_6DD8_Tx.Data[0]	:=	MCU_Rx.MCU_Thermal1_Rx.au8_Data[0];
ht_CAN4_6DD8_Tx.Data[1]	:=	MCU_Rx.MCU_Thermal1_Rx.au8_Data[1];
ht_CAN4_6DD8_Tx.Data[2]	:=	MCU_Rx.MCU_Thermal1_Rx.au8_Data[2];
ht_CAN4_6DD8_Tx.Data[3]	:=	MCU_Rx.MCU_Thermal1_Rx.au8_Data[3];
ht_CAN4_6DD8_Tx.Data[4]	:=	MCU_Rx.MCU_Thermal1_Rx.au8_Data[4];
ht_CAN4_6DD8_Tx.Data[5]	:=	MCU_Rx.MCU_Thermal1_Rx.au8_Data[5];
ht_CAN4_6DD8_Tx.Data[6]	:=	MCU_Rx.MCU_Thermal1_Rx.au8_Data[6];
ht_CAN4_6DD8_Tx.Data[7]	:=	MCU_Rx.MCU_Thermal1_Rx.au8_Data[7];
ht_CAN4_6DD8_Tx.Len		:=	8;


Tx_Timer(IN := NOT(Tx_Timer.Q), PT := T#1000MS);
IF (Tx_Timer.Q = TRUE) THEN
	
	G_CAN4_Channel.SendMessage(i_pMSG:=ADR(ht_CAN4_6DD0_Tx));
	G_CAN4_Channel.SendMessage(i_pMSG:=ADR(ht_CAN4_6DD1_Tx));
	G_CAN4_Channel.SendMessage(i_pMSG:=ADR(ht_CAN4_6DD2_Tx));
	G_CAN4_Channel.SendMessage(i_pMSG:=ADR(ht_CAN4_6DD3_Tx));
	G_CAN4_Channel.SendMessage(i_pMSG:=ADR(ht_CAN4_6DD4_Tx));
	G_CAN4_Channel.SendMessage(i_pMSG:=ADR(ht_CAN4_6DD5_Tx));
	G_CAN4_Channel.SendMessage(i_pMSG:=ADR(ht_CAN4_6DD6_Tx));
	G_CAN4_Channel.SendMessage(i_pMSG:=ADR(ht_CAN4_6DD7_Tx));
	G_CAN4_Channel.SendMessage(i_pMSG:=ADR(ht_CAN4_6DD8_Tx));
	END_IF

END_PROGRAM

// Application/UserCode/HMI/Data to or For HMI/Sevcon_to_HMI_1
PROGRAM Sevcon_to_HMI_1
VAR
	ht_CAN4_3DD0_Tx	:	EPEC_CANVXD.Msg;
	ht_CAN4_3DD1_Tx	:	EPEC_CANVXD.Msg;
	ht_CAN4_3DD2_Tx	:	EPEC_CANVXD.Msg;
	ht_CAN4_4DD0_Tx	:	EPEC_CANVXD.Msg;
	ht_CAN4_4DD1_Tx	:	EPEC_CANVXD.Msg;
	ht_CAN4_4DD2_Tx	:	EPEC_CANVXD.Msg;
	ht_CAN4_4DD3_Tx	:	EPEC_CANVXD.Msg;
	hton_MessageSend_Timer	:	TON;
	
	Tx_Timer	:	TON;
END_VAR


//*PowerSteering SEVCON
ht_CAN4_3DD0_Tx.ID		:=	16#183000DD OR EPEC_CANVXD.MASK_29BIT;
ht_CAN4_3DD0_Tx.Data[0]	:=	Sevcon_Steer_Rx.TorqueStatus1_Rx.au8_Data[0];
ht_CAN4_3DD0_Tx.Data[1]	:=	Sevcon_Steer_Rx.TorqueStatus1_Rx.au8_Data[1];
ht_CAN4_3DD0_Tx.Data[2]	:=	Sevcon_Steer_Rx.TorqueStatus1_Rx.au8_Data[2];
ht_CAN4_3DD0_Tx.Data[3]	:=	Sevcon_Steer_Rx.TorqueStatus1_Rx.au8_Data[3];
ht_CAN4_3DD0_Tx.Data[4]	:=	Sevcon_Steer_Rx.TorqueStatus1_Rx.au8_Data[4];
ht_CAN4_3DD0_Tx.Data[5]	:=	Sevcon_Steer_Rx.TorqueStatus1_Rx.au8_Data[5];
ht_CAN4_3DD0_Tx.Data[6]	:=	Sevcon_Steer_Rx.TorqueStatus1_Rx.au8_Data[6];
ht_CAN4_3DD0_Tx.Data[7]	:=	Sevcon_Steer_Rx.TorqueStatus1_Rx.au8_Data[7];
ht_CAN4_3DD0_Tx.Len		:=	8;

ht_CAN4_3DD1_Tx.ID		:=	16#183001DD OR EPEC_CANVXD.MASK_29BIT;
ht_CAN4_3DD1_Tx.Data[0]	:=	Sevcon_Steer_Rx.TorqueStatus2_Rx.au8_Data[0];
ht_CAN4_3DD1_Tx.Data[1]	:=	Sevcon_Steer_Rx.TorqueStatus2_Rx.au8_Data[1];
ht_CAN4_3DD1_Tx.Data[2]	:=	Sevcon_Steer_Rx.TorqueStatus2_Rx.au8_Data[2];
ht_CAN4_3DD1_Tx.Data[3]	:=	Sevcon_Steer_Rx.TorqueStatus2_Rx.au8_Data[3];
ht_CAN4_3DD1_Tx.Data[4]	:=	Sevcon_Steer_Rx.TorqueStatus2_Rx.au8_Data[4];
ht_CAN4_3DD1_Tx.Data[5]	:=	Sevcon_Steer_Rx.TorqueStatus2_Rx.au8_Data[5];
ht_CAN4_3DD1_Tx.Data[6]	:=	Sevcon_Steer_Rx.TorqueStatus2_Rx.au8_Data[6];
ht_CAN4_3DD1_Tx.Data[7]	:=	Sevcon_Steer_Rx.TorqueStatus2_Rx.au8_Data[7];
ht_CAN4_3DD1_Tx.Len		:=	8;

ht_CAN4_3DD2_Tx.ID		:=	16#183002DD OR EPEC_CANVXD.MASK_29BIT;
ht_CAN4_3DD2_Tx.Data[0]	:=	Sevcon_Steer_Rx.TempStatus_Rx.au8_Data[0];
ht_CAN4_3DD2_Tx.Data[1]	:=	Sevcon_Steer_Rx.TempStatus_Rx.au8_Data[1];
ht_CAN4_3DD2_Tx.Data[2]	:=	gu8_Sevcon1_Debug_Temp_Heatsink;
ht_CAN4_3DD2_Tx.Data[3]	:=	Sevcon_Steer_Rx.TempStatus_Rx.au8_Data[3];
ht_CAN4_3DD2_Tx.Data[4]	:=	Sevcon_Steer_Rx.TempStatus_Rx.au8_Data[4];
ht_CAN4_3DD2_Tx.Data[5]	:=	Sevcon_Steer_Rx.TempStatus_Rx.au8_Data[5];
ht_CAN4_3DD2_Tx.Data[6]	:=	Sevcon_Steer_Rx.TempStatus_Rx.au8_Data[6];
ht_CAN4_3DD2_Tx.Data[7]	:=	Sevcon_Steer_Rx.TempStatus_Rx.au8_Data[7];
ht_CAN4_3DD2_Tx.Len		:=	8;

(*Compressor SEVCON*)
ht_CAN4_4DD0_Tx.ID		:=	16#184000DD OR EPEC_CANVXD.MASK_29BIT;
ht_CAN4_4DD0_Tx.Data[0]	:=	Sevcon2_Rx.TorqueStatus1_Rx.au8_Data[0];
ht_CAN4_4DD0_Tx.Data[1]	:=	Sevcon2_Rx.TorqueStatus1_Rx.au8_Data[1];
ht_CAN4_4DD0_Tx.Data[2]	:=	Sevcon2_Rx.TorqueStatus1_Rx.au8_Data[2];
ht_CAN4_4DD0_Tx.Data[3]	:=	Sevcon2_Rx.TorqueStatus1_Rx.au8_Data[3];
ht_CAN4_4DD0_Tx.Data[4]	:=	Sevcon2_Rx.TorqueStatus1_Rx.au8_Data[4];
ht_CAN4_4DD0_Tx.Data[5]	:=	Sevcon2_Rx.TorqueStatus1_Rx.au8_Data[5];
ht_CAN4_4DD0_Tx.Data[6]	:=	Sevcon2_Rx.TorqueStatus1_Rx.au8_Data[6];
ht_CAN4_4DD0_Tx.Data[7]	:=	Sevcon2_Rx.TorqueStatus1_Rx.au8_Data[7];
ht_CAN4_4DD0_Tx.Len		:=	8;

ht_CAN4_4DD1_Tx.ID		:=	16#184001DD OR EPEC_CANVXD.MASK_29BIT;
ht_CAN4_4DD1_Tx.Data[0]	:=	Sevcon2_Rx.TorqueStatus2_Rx.au8_Data[0];
ht_CAN4_4DD1_Tx.Data[1]	:=	Sevcon2_Rx.TorqueStatus2_Rx.au8_Data[1];
ht_CAN4_4DD1_Tx.Data[2]	:=	Sevcon2_Rx.TorqueStatus2_Rx.au8_Data[2];
ht_CAN4_4DD1_Tx.Data[3]	:=	Sevcon2_Rx.TorqueStatus2_Rx.au8_Data[3];
ht_CAN4_4DD1_Tx.Data[4]	:=	Sevcon2_Rx.TorqueStatus2_Rx.au8_Data[4];
ht_CAN4_4DD1_Tx.Data[5]	:=	Sevcon2_Rx.TorqueStatus2_Rx.au8_Data[5];
ht_CAN4_4DD1_Tx.Data[6]	:=	Sevcon2_Rx.TorqueStatus2_Rx.au8_Data[6];
ht_CAN4_4DD1_Tx.Data[7]	:=	Sevcon2_Rx.TorqueStatus2_Rx.au8_Data[7];
ht_CAN4_4DD1_Tx.Len		:=	8;

ht_CAN4_4DD2_Tx.ID		:=	16#184002DD OR EPEC_CANVXD.MASK_29BIT;
ht_CAN4_4DD2_Tx.Data[0]	:=	Sevcon2_Rx.TempStatus_Rx.au8_Data[0];
ht_CAN4_4DD2_Tx.Data[1]	:=	Sevcon2_Rx.TempStatus_Rx.au8_Data[1];
ht_CAN4_4DD2_Tx.Data[2]	:=	Sevcon2_Rx.TempStatus_Rx.au8_Data[2];
ht_CAN4_4DD2_Tx.Data[3]	:=	Sevcon2_Rx.TempStatus_Rx.au8_Data[3];
ht_CAN4_4DD2_Tx.Data[4]	:=	Sevcon2_Rx.TempStatus_Rx.au8_Data[4];
ht_CAN4_4DD2_Tx.Data[5]	:=	Sevcon2_Rx.TempStatus_Rx.au8_Data[5];
ht_CAN4_4DD2_Tx.Data[6]	:=	Sevcon2_Rx.TempStatus_Rx.au8_Data[6];
ht_CAN4_4DD2_Tx.Data[7]	:=	Sevcon2_Rx.TempStatus_Rx.au8_Data[7];
ht_CAN4_4DD2_Tx.Len		:=	8;

ht_CAN4_4DD3_Tx.ID		:=	16#184003DD OR EPEC_CANVXD.MASK_29BIT;
ht_CAN4_4DD3_Tx.Data[0]	:=	Sevcon2_Rx.Compressor_Temp_Rx.au8_Data[5];
ht_CAN4_4DD3_Tx.Data[1]	:=	Sevcon2_Rx.Compressor_Temp_Rx.au8_Data[6];
ht_CAN4_4DD3_Tx.Data[2]	:=	gu8_Sevcon1_Debug_Temp_Heatsink;
ht_CAN4_4DD3_Tx.Data[3].0	:= Sevcon2_Control.NO_OIL;
ht_CAN4_4DD3_Tx.Data[3].1	:= Sevcon2_Rx.Compressor_Oil_Rx.au8_Data[2].4;
ht_CAN4_4DD3_Tx.Data[3].2	:= Sevcon2_Control.Oil_Level_Warning;
ht_CAN4_4DD3_Tx.Data[3].3	:= Sevcon2_Control.Compressor_Temp_Warning;
ht_CAN4_4DD3_Tx.Data[3].4	:= Sevcon2_Control.Compressor_Temp_Fault;
ht_CAN4_4DD3_Tx.Data[3].5	:= Sevcon2_Control.Air_Temp_Warning;
ht_CAN4_4DD3_Tx.Data[3].6	:= Sevcon2_Control.Air_Temp_Fault;
ht_CAN4_4DD3_Tx.Data[3].7	:= CAN1_Rx.Bob_J1939_AirPressure_Rx.au8_Data[6].0;
ht_CAN4_4DD3_Tx.Data[4]	:=	16#00;
ht_CAN4_4DD3_Tx.Data[5]	:=	16#00;
ht_CAN4_4DD3_Tx.Data[6]	:=	16#00;
ht_CAN4_4DD3_Tx.Data[7]	:=	16#00;
ht_CAN4_4DD3_Tx.Len		:=	8;


Tx_Timer(IN := NOT(Tx_Timer.Q), PT := T#1000MS);
IF (Tx_Timer.Q = TRUE) THEN
	G_CAN4_Channel.SendMessage(i_pMSG:=ADR(ht_CAN4_3DD0_Tx));
	G_CAN4_Channel.SendMessage(i_pMSG:=ADR(ht_CAN4_3DD1_Tx));
	G_CAN4_Channel.SendMessage(i_pMSG:=ADR(ht_CAN4_3DD2_Tx));
	G_CAN4_Channel.SendMessage(i_pMSG:=ADR(ht_CAN4_4DD0_Tx));
	G_CAN4_Channel.SendMessage(i_pMSG:=ADR(ht_CAN4_4DD1_Tx));
	G_CAN4_Channel.SendMessage(i_pMSG:=ADR(ht_CAN4_4DD2_Tx));
	G_CAN4_Channel.SendMessage(i_pMSG:=ADR(ht_CAN4_4DD3_Tx));

END_IF

END_PROGRAM

// Application/UserCode/HMI/Data to or For HMI/VMU_to_HMI_1
PROGRAM VMU_to_HMI_1
VAR
	CAN4_VMU0_Tx			:	EPEC_CANVXD.Msg;	// Digital
	CAN4_VMU1_Tx			: 	EPEC_CANVXD.Msg;	// Digital
	CAN4_VMU2_Tx			: 	EPEC_CANVXD.Msg;
	CAN4_VMU3_Tx			: 	EPEC_CANVXD.Msg;
	CAN4_VMU4_Tx			: 	EPEC_CANVXD.Msg;
	CAN4_VMU5_Tx			: 	EPEC_CANVXD.Msg;
	hton_MessageSend_Timer	:	TON;
	Tx_Timer				:	TON;
END_VAR

//called from can4_TX
// Connector C1 DIGITAL ONLY
CAN4_VMU0_Tx.ID			:=	16#190000DD OR EPEC_CANVXD.MASK_29BIT;
CAN4_VMU0_Tx.Len		:= 8;
CAN4_VMU0_Tx.Data[0].0	:= DI_q_Spare_X1_11_DI;							//Pin 1.11 - Filtered digital input status.
CAN4_VMU0_Tx.Data[0].1	:= DOS_q_BackupPump_DO;							//X1.12 Backup power steering
CAN4_VMU0_Tx.Data[0].2	:= DO_q_BackupPump_DO; 							//X1.12 Backup power steering
CAN4_VMU0_Tx.Data[0].3	:= DOS_q_BatteryDischargeMain_DO; 				//X1.22 Battery Discharge Main
CAN4_VMU0_Tx.Data[0].4	:= DO_q_BatteryDischargeMain_DO;  				//X1.22 Battery Discharge Main
CAN4_VMU0_Tx.Data[0].5	:= DOS_q_ePTO_Fan_DO; 							//X1.23 ePTO Fan Enable
CAN4_VMU0_Tx.Data[0].6	:= DO_q_ePTO_Fan_DO;							//X1.23 ePTO Fan Enable
CAN4_VMU0_Tx.Data[0].7  := DOS_q_Battery1ChargePrecharge_DO;			//X1.29 Soft Charge Battery 1
CAN4_VMU0_Tx.Data[1].0  := DO_q_Battery1ChargePrecharge_DO;				//X1.29 Soft Charge Battery 1
CAN4_VMU0_Tx.Data[1].1  := DOS_q_Battery1ChargeMain_DO; 				//X1.30 Charge Main Battery 1
CAN4_VMU0_Tx.Data[1].2  := DO_q_Battery1ChargeMain_DO;					//Pin 1.30 - Digital output status for output pin. 
CAN4_VMU0_Tx.Data[1].3  := DOS_q_Battery2ChargePrecharge_DO; 			//X1.31 Soft Charge Battery 2
CAN4_VMU0_Tx.Data[1].4  := DO_q_Battery2ChargePrecharge_DO;				//X1.31 Soft Charge Battery 2
CAN4_VMU0_Tx.Data[1].5  := DOS_q_DrivetrainInverterTorqueless_DO;		//Pin 1.32 - Digital input state for pin.	
CAN4_VMU0_Tx.Data[1].6  := DO_q_DrivetrainInverterTorqueless_DO;		//Pin 1.32 - Digital output status for output pin.
CAN4_VMU0_Tx.Data[1].7  := DOS_q_BatteryDischargePrecharge_DO; 			//X1.33 Soft Discharge Battery 1
CAN4_VMU0_Tx.Data[2].0  := DO_q_BatteryDischargePrecharge_DO;			//Pin 1.33 - Digital output status for output pin. 
CAN4_VMU0_Tx.Data[2].1  := DOS_q_Battery2ChargeMain_DO; 				//X1.35 Charge Main Battery 2
CAN4_VMU0_Tx.Data[2].2  := DO_q_Battery2ChargeMain_DO;					//Pin 1.35 - Digital output status for output pin.
// Connector C2 DIGITAL ONLY
CAN4_VMU0_Tx.Data[2].3  := DI_q_Aux_Pos_Discharge_Master_DI; 			//Pin 2.6 - Filtered digital input status.
CAN4_VMU0_Tx.Data[2].4  := DI_q_Aux_Neg_Discharge_Master_DI; 			//Pin 2.7 - Filtered digital input status.
CAN4_VMU0_Tx.Data[2].5  := DI_q_Aux_Pos_Discharge_Slave_DI; 			//Pin 2.8 - Filtered digital input status.
CAN4_VMU0_Tx.Data[2].6  := DI_q_Aux_Neg_Discharge_Slave_DI; 			//Pin 2.9 - Filtered digital input status.
CAN4_VMU0_Tx.Data[2].7  := DOS_q_ChargePlugLockPulse_DO ; 				//Pin 2.13 - Digital input state for pin.
CAN4_VMU0_Tx.Data[3].0  := DO_q_ChargePlugLockPulse_DO;					//Pin 2.13 - Digital output status for output pin.
CAN4_VMU0_Tx.Data[3].1  := DOS_q_ChargePlugLockPosition_DO; 			//Pin 2.14 - Digital input state for pin.
CAN4_VMU0_Tx.Data[3].2  := DO_q_ChargePlugLockPosition_DO;				//Pin 2.14 - Digital output status for output pin.
CAN4_VMU0_Tx.Data[3].3  := DI_q_PB_Cruise_Control_DI; 				//Pin 2.16 - Filtered digital input status.
CAN4_VMU0_Tx.Data[3].4  := DOS_q_DrivetrainKL15D_DO; 					//Pin 2.28 - Digital input state for pin.
CAN4_VMU0_Tx.Data[3].5  := DO_q_DrivetrainKL15D_DO;						//Pin 2.28 - Digital output status for output pin.
CAN4_VMU0_Tx.Data[3].6  := DOS_q_DrivetrainKL15C_DO; 					//Pin 2.29 - Digital input state for pin.
CAN4_VMU0_Tx.Data[3].7  := DO_q_DrivetrainKL15C_DO;						//Pin 2.29 - Digital output status for output pin.
CAN4_VMU0_Tx.Data[4].0  := DOS_q_DrivetrainCoolingFan_DO; 				//Pin 2.30 - Digital input state for pin.
CAN4_VMU0_Tx.Data[4].1  := DO_q_DrivetrainCoolingFan_DO;				//Pin 2.30 - Digital output status for output pin.
CAN4_VMU0_Tx.Data[4].2  := DOS_q_DrievtrainPowerSteering_DO; 			//Pin 2.31 - Digital input state for pin.
CAN4_VMU0_Tx.Data[4].3  := DO_q_DrievtrainPowerSteering_DO;				//Pin 2.31 - Digital output status for output pin.
CAN4_VMU0_Tx.Data[4].4  := DOS_q_Sw_Body_Step_DO; 			//Pin 2.33 - Digital input state for pin.
CAN4_VMU0_Tx.Data[4].5  := DO_q_Sw_Body_Step_DO;				//Pin 2.33 - Digital output status for output pin.
CAN4_VMU0_Tx.Data[4].6  := DOS_q_DynamoD_DO; 							//Pin 2.35 - Digital input state for pin.
CAN4_VMU0_Tx.Data[4].7  := DO_q_DynamoD_DO;								//Pin 2.35 - Digital output state for sinking digital output.
// Connector C3 DIGITAL ONLY
CAN4_VMU0_Tx.Data[5].0  := DI_q_PB_E_Stop_OK_DI; 		//Pin 3.5 - Filtered digital input status.
CAN4_VMU0_Tx.Data[5].1  := DI_q_DirectionSwitch_Drive_DI; 				//Pin 3.6 - Filtered digital input status.
CAN4_VMU0_Tx.Data[5].2  := DI_q_IlluminiationStatsus_DI; 				//Pin 3.7 - Filtered digital input status.
CAN4_VMU0_Tx.Data[5].3  := DI_q_DirectionSwitch_Reverse_DI; 			//Pin 3.8 - Filtered digital input status.
CAN4_VMU0_Tx.Data[5].4  := DI_q_DirectionSwitch_DriveCrawl_DI; 			//Pin 3.9 - Filtered digital input status.
CAN4_VMU0_Tx.Data[5].5  := DI_q_DirectionSwitch_Neutral_DI; 			//Pin 3.11 - Filtered digital input status.
CAN4_VMU0_Tx.Data[5].6  := DI_q_VehicleKL15_DI; 						//Pin 3.22 - Filtered digital input status.
CAN4_VMU0_Tx.Data[5].7  := DI_q_VehicleKL51_DI; 						//Pin 3.23 - Filtered digital input status.
CAN4_VMU0_Tx.Data[6].0  := DOS_q_ChargersWakeup_DO; 					//Pin 3.26 - Digital input state for pin.
CAN4_VMU0_Tx.Data[6].1  := DO_q_ChargersWakeup_DO;						//Pin 3.26 - Digital output status for output pin.
CAN4_VMU0_Tx.Data[6].2  := DOS_q_DashboardDCDCStatus_DO; 				//Pin 3.27 - Digital input state for pin.
CAN4_VMU0_Tx.Data[6].3  := DO_q_DashboardDCDCStatus_DO;					//Pin 3.27 - Digital output status for output pin.
CAN4_VMU0_Tx.Data[6].4  := DI_q_HeaterIn_DI; 							//Pin 3.28 - Filtered digital input status.
CAN4_VMU0_Tx.Data[6].5  := DOS_q_HeaterOut_DI; 							//Pin 3.29 - Digital input state for pin.
CAN4_VMU0_Tx.Data[6].6  := DO_q_HeaterOut_DI;							//Pin 3.29 - Digital output status for output pin.
CAN4_VMU0_Tx.Data[6].7  := DOS_q_DrivetrainInverterRf1_DO; 				//Pin 3.30 - Digital input state for pin.
CAN4_VMU0_Tx.Data[7].0  := DO_q_DrivetrainInverterRf1_DO;				//Pin 3.30 - Digital output status for output pin.	
CAN4_VMU0_Tx.Data[7].1  := DOS_q_DrivetrainInverterRf2_DO; 				//Pin 3.31 - Digital input state for pin.
CAN4_VMU0_Tx.Data[7].2  := DO_q_DrivetrainInverterRf2_DO;				//Pin 3.31 - Digital output status for output pin.
CAN4_VMU0_Tx.Data[7].3  := DOS_q_DrivetrainDCDCInhibit_DO; 				//Pin 3.32 - Digital input state for pin.
CAN4_VMU0_Tx.Data[7].4  := DO_q_DrivetrainDCDCInhibit_DO;				//Pin 3.32 - Digital output status for output pin.
CAN4_VMU0_Tx.Data[7].5  := DOS_q_ChargePlugLED_Green_DO; 				//Pin 3.33 - Digital input state for pin.
CAN4_VMU0_Tx.Data[7].6  := DO_q_ChargePlugLED_Green_DO;					//Pin 3.33 - Digital output status for output pin.
CAN4_VMU0_Tx.Data[7].7  := DOS_q_ChargePlugLED_Blue_DO; 				//Pin 3.34 - Digital input state for pin.

// Connector C3 DIGITAL ONLY Continued
CAN4_VMU1_Tx.ID			:=	16#190001DD OR EPEC_CANVXD.MASK_29BIT;
CAN4_VMU1_Tx.Len		:= 8;
CAN4_VMU1_Tx.Data[0].0  := DO_q_ChargePlugLED_Blue_DO;					//Pin 3.34 - Digital output status for output pin.
CAN4_VMU1_Tx.Data[0].1  := DOS_q_ChargePlugLED_Red_DO; 					//Pin 3.35 - Digital input state for pin.
CAN4_VMU1_Tx.Data[0].2  := DO_q_ChargePlugLED_Red_DO;					//Pin 3.35 - Digital output status for output pin.
CAN4_VMU1_Tx.Data[0].3  := 0;											//Spare.
//Ditto																	//Ditto.

//Anal Stuff
CAN4_VMU2_Tx.ID			:=	16#190002DD OR EPEC_CANVXD.MASK_29BIT;
CAN4_VMU2_Tx.Len		:= 8;
CAN4_VMU2_Tx.Data[0]	:=	WORD_TO_BYTE 	(AIPU_u16_KEB_Temperature_Sensor_AI);				//Pin 1.9 - Filtered AI value
CAN4_VMU2_Tx.Data[1]	:=	WORD_TO_BYTE 	(SHR (AIPU_u16_KEB_Temperature_Sensor_AI, 8));		//Pin 1.9 - Filtered AI value
CAN4_VMU2_Tx.Data[2]	:=	WORD_TO_BYTE 	(AI_u16_KEB_Temperature_Sensor_AI);					//Pin 1.9 - Filtered AI value
CAN4_VMU2_Tx.Data[3]	:=	WORD_TO_BYTE 	(SHR (AI_u16_KEB_Temperature_Sensor_AI, 8));		//Pin 1.9 - Filtered AI value
CAN4_VMU2_Tx.Data[4]	:=	WORD_TO_BYTE 	(AIPU_u16_Spare_X1_10_AI);			//Pin 1.10 - Filtered AI value
CAN4_VMU2_Tx.Data[5]	:=	WORD_TO_BYTE 	(SHR (AIPU_u16_Spare_X1_10_AI, 8)); 	//Pin 1.10 - Filtered AI value
CAN4_VMU2_Tx.Data[6]	:=	WORD_TO_BYTE 	(AI_u16_Spare_X1_10_AI);				//Pin 1.10 - Filtered AI value
CAN4_VMU2_Tx.Data[7]	:=	WORD_TO_BYTE 	(SHR (AI_u16_Spare_X1_10_AI, 8));		//Pin 1.10 - Filtered AI value

CAN4_VMU3_Tx.ID			:=	16#190003DD OR EPEC_CANVXD.MASK_29BIT;
CAN4_VMU3_Tx.Len		:= 8;
CAN4_VMU3_Tx.Data[0]	:=	WORD_TO_BYTE 	(AIPU_u16_Heater1Temperature_AI);			//Pin 1.20 - Filtered AI value
CAN4_VMU3_Tx.Data[1]	:=	WORD_TO_BYTE 	(SHR (AIPU_u16_Heater1Temperature_AI, 8));	//Pin 1.20 - Filtered AI value
CAN4_VMU3_Tx.Data[2]	:=	WORD_TO_BYTE 	(AI_u16_Heater1Temperature_AI);				//Pin 1.20 - Filtered AI value
CAN4_VMU3_Tx.Data[3]	:=	WORD_TO_BYTE 	(SHR (AI_u16_Heater1Temperature_AI, 8));	//Pin 1.20 - Filtered AI value
CAN4_VMU3_Tx.Data[4]	:=	WORD_TO_BYTE 	(AIPU_u16_Heater2Temperature_AI);			//Pin 1.21 - Filtered AI value
CAN4_VMU3_Tx.Data[5]	:=	WORD_TO_BYTE 	(SHR (AIPU_u16_Heater2Temperature_AI, 8));	//Pin 1.21 - Filtered AI value
CAN4_VMU3_Tx.Data[6]	:=	WORD_TO_BYTE 	(AI_u16_Heater2Temperature_AI);				//Pin 1.21 - Filtered AI value
CAN4_VMU3_Tx.Data[7]	:=	WORD_TO_BYTE 	(SHR (AI_u16_Heater2Temperature_AI, 8));	//Pin 1.21 - Filtered AI value

CAN4_VMU4_Tx.ID			:=	16#190004DD OR EPEC_CANVXD.MASK_29BIT;	
CAN4_VMU4_Tx.Len		:= 8;					
CAN4_VMU4_Tx.Data[0]	:=	WORD_TO_BYTE 	(AIPU_u16_HeaterDiagnose_AI);				//Pin 2.23 - Filtered AI value
CAN4_VMU4_Tx.Data[1]	:=	WORD_TO_BYTE 	(SHR (AIPU_u16_HeaterDiagnose_AI, 8));		//Pin 2.23 - Filtered AI value
CAN4_VMU4_Tx.Data[2]	:=	WORD_TO_BYTE 	(AI_u16_HeaterDiagnose_AI);					//Pin 2.23 - Filtered AI value
CAN4_VMU4_Tx.Data[3]	:=	WORD_TO_BYTE 	(SHR (AI_u16_HeaterDiagnose_AI, 8));		//Pin 2.23 - Filtered AI value
CAN4_VMU4_Tx.Data[4]	:=	WORD_TO_BYTE 	(AIPU_u16_HeaterDiagnose2_AI);				//Pin 3.14 - Filtered AI value
CAN4_VMU4_Tx.Data[5]	:=	WORD_TO_BYTE 	(SHR (AIPU_u16_HeaterDiagnose2_AI, 8));		//Pin 3.14 - Filtered AI value
CAN4_VMU4_Tx.Data[6]	:=	WORD_TO_BYTE 	(AI_u16_Heater1Temperature_AI);				//Pin 3.14 - Filtered AI value
CAN4_VMU4_Tx.Data[7]	:=	WORD_TO_BYTE 	(SHR (AI_u16_Heater1Temperature_AI, 8));	//Pin 3.14 - Filtered AI value

CAN4_VMU5_Tx.ID			:=	16#190005DD OR EPEC_CANVXD.MASK_29BIT;
CAN4_VMU5_Tx.Len		:= 8;
CAN4_VMU5_Tx.Data[0]	:=	WORD_TO_BYTE 	(AIPU_u16_VehicleThrottlePedal1_AI);		//Pin 3.15 - Filtered AI value
CAN4_VMU5_Tx.Data[1]	:=	WORD_TO_BYTE 	(SHR(AIPU_u16_VehicleThrottlePedal1_AI,8)); //Pin 3.15 - Filtered AI value
CAN4_VMU5_Tx.Data[2]	:=	WORD_TO_BYTE 	(AI_u16_VehicleThrottlePedal1_AI);			//Pin 3.15 - Filtered AI value
CAN4_VMU5_Tx.Data[3]	:=	WORD_TO_BYTE 	(SHR (AI_u16_VehicleThrottlePedal1_AI,8));	//Pin 3.15 - Filtered AI value
CAN4_VMU5_Tx.Data[4]	:=	WORD_TO_BYTE 	(AIPU_u16_VehicleThrottlePedal2_AI	);		//Pin 3.16 - Filtered AI value 
CAN4_VMU5_Tx.Data[5]	:=	WORD_TO_BYTE 	(SHR(AIPU_u16_VehicleThrottlePedal2_AI,8)); //Pin 3.16 - Filtered AI value 
CAN4_VMU5_Tx.Data[6]	:=	WORD_TO_BYTE 	(AI_u16_VehicleThrottlePedal2_AI);			//Pin 3.16 - Filtered AI value 
CAN4_VMU5_Tx.Data[7]	:=	WORD_TO_BYTE 	(SHR(AI_u16_VehicleThrottlePedal2_AI, 8));	//Pin 3.16 - Filtered AI value 


Tx_Timer(IN := NOT(Tx_Timer.Q), PT := T#100MS);
IF (Tx_Timer.Q = TRUE) THEN
	G_CAN4_Channel.SendMessage(i_pMSG:=ADR(CAN4_VMU0_Tx));
	G_CAN4_Channel.SendMessage(i_pMSG:=ADR(CAN4_VMU1_Tx));
	G_CAN4_Channel.SendMessage(i_pMSG:=ADR(CAN4_VMU2_Tx));
	G_CAN4_Channel.SendMessage(i_pMSG:=ADR(CAN4_VMU3_Tx));
	G_CAN4_Channel.SendMessage(i_pMSG:=ADR(CAN4_VMU4_Tx));
	G_CAN4_Channel.SendMessage(i_pMSG:=ADR(CAN4_VMU5_Tx));
END_IF

END_PROGRAM

// Application/UserCode/BMS/CATL/CATLBMS1_Rx
PROGRAM CATLBMS1_Rx

(*Program to receive all data from the CATL BMS*)



(*Initial saving CAN messages to receipt strucutres*)


(*Unpacking structures into variables*)


(*Comms loss check to ensure all messages are still being received*)


CATLBMS_RxConversion();

END_PROGRAM

// Application/UserCode/CAN Function Blocks/CAN2/Callback_Receive_CAN2
FUNCTION_BLOCK Callback_Receive_CAN2 IMPLEMENTS
EPEC_CANVXD.IReceiveCallback
VAR_INPUT	
END_VAR
VAR_OUTPUT
END_VAR
VAR
END_VAR

METHOD Receive
VAR_INPUT
	(* Pointer to the CAN message *)
	i_pMsg	: POINTER TO EPEC_CANVXD.Msg;
	(* User specific argument. This is set in AddCOBID i_Argument. *)
	i_Argument	: DWORD;
END_VAR
VAR
	t_pRxMessage : POINTER TO t_CANReceive;
END_VAR


t_pRxMessage				:=	i_Argument;
t_pRxMessage^.q_NewDataRxed	:=	TRUE;
t_pRxMessage^.Data			:=	i_pMsg^.Data;
t_pRxMessage^.ID			:=	i_pMsg^.ID;
t_pRxMessage^.Len			:=	i_pMsg^.Len;
END_METHOD

END_FUNCTION_BLOCK

// Application/UserCode/CAN Function Blocks/CAN3/Callback_Receive_CAN3
FUNCTION_BLOCK Callback_Receive_CAN3 IMPLEMENTS
EPEC_CANVXD.IReceiveCallback
VAR_INPUT	
END_VAR
VAR_OUTPUT
END_VAR
VAR
END_VAR

METHOD Receive
VAR_INPUT
	(* Pointer to the CAN message *)
	i_pMsg	: POINTER TO EPEC_CANVXD.Msg;
	(* User specific argument. This is set in AddCOBID i_Argument. *)
	i_Argument	: DWORD;
END_VAR
VAR
	t_pRxMessage : POINTER TO t_CANReceive;
END_VAR


t_pRxMessage				:=	i_Argument;
t_pRxMessage^.q_NewDataRxed	:=	TRUE;
t_pRxMessage^.Data			:=	i_pMsg^.Data;
t_pRxMessage^.ID			:=	i_pMsg^.ID;
t_pRxMessage^.Len			:=	i_pMsg^.Len;
END_METHOD

END_FUNCTION_BLOCK

// Application/UserCode/CAN Function Blocks/CAN4/Callback_Receive_CAN4
FUNCTION_BLOCK Callback_Receive_CAN4 IMPLEMENTS
EPEC_CANVXD.IReceiveCallback
VAR_INPUT	
END_VAR
VAR_OUTPUT
END_VAR
VAR
END_VAR

METHOD Receive
VAR_INPUT
	(* Pointer to the CAN message *)
	i_pMsg	: POINTER TO EPEC_CANVXD.Msg;
	(* User specific argument. This is set in AddCOBID i_Argument. *)
	i_Argument	: DWORD;
END_VAR
VAR
	t_pRxMessage : POINTER TO t_CANReceive;
END_VAR


t_pRxMessage				:=	i_Argument;
t_pRxMessage^.q_NewDataRxed	:=	TRUE;
t_pRxMessage^.Data			:=	i_pMsg^.Data;
t_pRxMessage^.ID			:=	i_pMsg^.ID;
t_pRxMessage^.Len			:=	i_pMsg^.Len;
END_METHOD

END_FUNCTION_BLOCK
